LIN{ E6POS: X 709.1620, Y 12.2455, Z -112.0150, A 0, B 90, C 0, E1 0, E2 0, E3 0, E4 0 } C_DIS
LIN{ E6POS: X 709.1855, Y 12.9576, Z -112.0150, A 0, B 90, C 0, E1 0, E2 0, E3 0, E4 0 } C_DIS
LIN{ E6POS: X 709.1944, Y 13.6424, Z -112.0150, A 0, B 90, C 0, E1 0, E2 0, E3 0, E4 0 } C_DIS
LIN{ E6POS: X 709.2185, Y 14.3759, Z -112.0150, A 0, B 90, C 0, E1 0, E2 0, E3 0, E4 0 } C_DIS
LIN{ E6POS: X 709.2277, Y 15.0601, Z -112.0150, A 0, B 90, C 0, E1 0, E2 0, E3 0, E4 0 } C_DIS
LIN{ E6POS: X 709.2521, Y 15.7930, Z -112.0150, A 0, B 90, C 0, E1 0, E2 0, E3 0, E4 0 } C_DIS
LIN{ E6POS: X 709.2586, Y 16.4546, Z -112.0150, A 0, B 90, C 0, E1 0, E2 0, E3 0, E4 0 } C_DIS
LIN{ E6POS: X 709.2824, Y 17.1639, Z -112.0150, A 0, B 90, C 0, E1 0, E2 0, E3 0, E4 0 } C_DIS
LIN{ E6POS: X 709.2841, Y 17.7821, Z -112.0150, A 0, B 90, C 0, E1 0, E2 0, E3 0, E4 0 } C_DIS
LIN{ E6POS: X 709.3065, Y 18.4443, Z -112.0150, A 0, B 90, C 0, E1 0, E2 0, E3 0, E4 0 } C_DIS
LIN{ E6POS: X 709.3061, Y 19.0402, Z -112.0150, A 0, B 90, C 0, E1 0, E2 0, E3 0, E4 0 } C_DIS
LIN{ E6POS: X 709.3272, Y 19.6784, Z -112.0150, A 0, B 90, C 0, E1 0, E2 0, E3 0, E4 0 } C_DIS
LIN{ E6POS: X 709.3275, Y 20.2736, Z -112.0150, A 0, B 90, C 0, E1 0, E2 0, E3 0, E4 0 } C_DIS
LIN{ E6POS: X 709.3493, Y 20.9106, Z -112.0150, A 0, B 90, C 0, E1 0, E2 0, E3 0, E4 0 } C_DIS
LIN{ E6POS: X 709.3528, Y 21.5252, Z -112.0150, A 0, B 90, C 0, E1 0, E2 0, E3 0, E4 0 } C_DIS
LIN{ E6POS: X 709.3767, Y 22.1837, Z -112.0150, A 0, B 90, C 0, E1 0, E2 0, E3 0, E4 0 } C_DIS
LIN{ E6POS: X 709.3863, Y 22.8398, Z -112.0150, A 0, B 90, C 0, E1 0, E2 0, E3 0, E4 0 } C_DIS
LIN{ E6POS: X 709.4122, Y 23.5420, Z -112.0150, A 0, B 90, C 0, E1 0, E2 0, E3 0, E4 0 } C_DIS
LIN{ E6POS: X 709.4258, Y 24.1924, Z -112.0150, A 0, B 90, C 0, E1 0, E2 0, E3 0, E4 0 } C_DIS
LIN{ E6POS: X 709.4549, Y 24.8978, Z -112.0150, A 0, B 90, C 0, E1 0, E2 0, E3 0, E4 0 } C_DIS
LIN{ E6POS: X 709.4716, Y 25.4954, Z -112.0150, A 0, B 90, C 0, E1 0, E2 0, E3 0, E4 0 } C_DIS
LIN{ E6POS: X 709.5021, Y 26.1621, Z -112.0150, A 0, B 90, C 0, E1 0, E2 0, E3 0, E4 0 } C_DIS
LIN{ E6POS: X 709.5463, Y 27.1611, Z -112.0150, A 0, B 90, C 0, E1 0, E2 0, E3 0, E4 0 } C_DIS
LIN{ E6POS: X 709.5464, Y 27.1641, Z -112.0150, A 0, B 90, C 0, E1 0, E2 0, E3 0, E4 0 } C_DIS
LIN{ E6POS: X 709.6142, Y 28.1618, Z -112.0150, A 0, B 90, C 0, E1 0, E2 0, E3 0, E4 0 } C_DIS
LIN{ E6POS: X 709.6325, Y 28.4296, Z -112.0150, A 0, B 90, C 0, E1 0, E2 0, E3 0, E4 0 } C_DIS
LIN{ E6POS: X 709.6724, Y 29.4288, Z -112.0150, A 0, B 90, C 0, E1 0, E2 0, E3 0, E4 0 } C_DIS
LIN{ E6POS: X 709.6727, Y 29.4368, Z -112.0150, A 0, B 90, C 0, E1 0, E2 0, E3 0, E4 0 } C_DIS
LIN{ E6POS: X 709.7423, Y 30.4344, Z -112.0150, A 0, B 90, C 0, E1 0, E2 0, E3 0, E4 0 } C_DIS
LIN{ E6POS: X 709.7598, Y 30.6853, Z -112.0150, A 0, B 90, C 0, E1 0, E2 0, E3 0, E4 0 } C_DIS
LIN{ E6POS: X 709.7733, Y 31.4340, Z -112.0150, A 0, B 90, C 0, E1 0, E2 0, E3 0, E4 0 } C_DIS
LIN{ E6POS: X 709.8048, Y 32.1998, Z -112.0150, A 0, B 90, C 0, E1 0, E2 0, E3 0, E4 0 } C_DIS
LIN{ E6POS: X 709.8180, Y 33.0718, Z -112.0150, A 0, B 90, C 0, E1 0, E2 0, E3 0, E4 0 } C_DIS
LIN{ E6POS: X 709.8486, Y 33.9336, Z -112.0150, A 0, B 90, C 0, E1 0, E2 0, E3 0, E4 0 } C_DIS
LIN{ E6POS: X 709.8618, Y 34.8057, Z -112.0150, A 0, B 90, C 0, E1 0, E2 0, E3 0, E4 0 } C_DIS
LIN{ E6POS: X 709.8928, Y 35.6668, Z -112.0150, A 0, B 90, C 0, E1 0, E2 0, E3 0, E4 0 } C_DIS
LIN{ E6POS: X 709.9072, Y 36.4152, Z -112.0150, A 0, B 90, C 0, E1 0, E2 0, E3 0, E4 0 } C_DIS
LIN{ E6POS: X 709.9403, Y 37.1800, Z -112.0150, A 0, B 90, C 0, E1 0, E2 0, E3 0, E4 0 } C_DIS
LIN{ E6POS: X 709.9764, Y 38.0568, Z -112.0150, A 0, B 90, C 0, E1 0, E2 0, E3 0, E4 0 } C_DIS
LIN{ E6POS: X 710.0507, Y 39.0541, Z -112.0150, A 0, B 90, C 0, E1 0, E2 0, E3 0, E4 0 } C_DIS
LIN{ E6POS: X 710.0543, Y 39.1022, Z -112.0150, A 0, B 90, C 0, E1 0, E2 0, E3 0, E4 0 } C_DIS
LIN{ E6POS: X 710.1008, Y 39.9703, Z -112.0150, A 0, B 90, C 0, E1 0, E2 0, E3 0, E4 0 } C_DIS
LIN{ E6POS: X 710.1840, Y 40.9668, Z -112.0150, A 0, B 90, C 0, E1 0, E2 0, E3 0, E4 0 } C_DIS
LIN{ E6POS: X 710.1874, Y 41.0075, Z -112.0150, A 0, B 90, C 0, E1 0, E2 0, E3 0, E4 0 } C_DIS
LIN{ E6POS: X 710.2166, Y 41.7433, Z -112.0150, A 0, B 90, C 0, E1 0, E2 0, E3 0, E4 0 } C_DIS
LIN{ E6POS: X 710.2637, Y 42.4956, Z -112.0150, A 0, B 90, C 0, E1 0, E2 0, E3 0, E4 0 } C_DIS
LIN{ E6POS: X 710.2954, Y 43.3763, Z -112.0150, A 0, B 90, C 0, E1 0, E2 0, E3 0, E4 0 } C_DIS
LIN{ E6POS: X 710.3438, Y 44.2406, Z -112.0150, A 0, B 90, C 0, E1 0, E2 0, E3 0, E4 0 } C_DIS
LIN{ E6POS: X 710.3760, Y 45.1706, Z -112.0150, A 0, B 90, C 0, E1 0, E2 0, E3 0, E4 0 } C_DIS
LIN{ E6POS: X 710.4250, Y 46.0693, Z -112.0150, A 0, B 90, C 0, E1 0, E2 0, E3 0, E4 0 } C_DIS
LIN{ E6POS: X 710.4558, Y 46.9518, Z -112.0150, A 0, B 90, C 0, E1 0, E2 0, E3 0, E4 0 } C_DIS
LIN{ E6POS: X 710.5046, Y 47.8100, Z -112.0150, A 0, B 90, C 0, E1 0, E2 0, E3 0, E4 0 } C_DIS
LIN{ E6POS: X 710.5328, Y 48.5487, Z -112.0150, A 0, B 90, C 0, E1 0, E2 0, E3 0, E4 0 } C_DIS
LIN{ E6POS: X 710.5811, Y 49.2887, Z -112.0150, A 0, B 90, C 0, E1 0, E2 0, E3 0, E4 0 } C_DIS
LIN{ E6POS: X 710.6062, Y 49.9190, Z -112.0150, A 0, B 90, C 0, E1 0, E2 0, E3 0, E4 0 } C_DIS
LIN{ E6POS: X 710.6544, Y 50.5709, Z -112.0150, A 0, B 90, C 0, E1 0, E2 0, E3 0, E4 0 } C_DIS
LIN{ E6POS: X 710.6788, Y 51.1296, Z -112.0150, A 0, B 90, C 0, E1 0, E2 0, E3 0, E4 0 } C_DIS
LIN{ E6POS: X 710.7266, Y 51.7228, Z -112.0150, A 0, B 90, C 0, E1 0, E2 0, E3 0, E4 0 } C_DIS
LIN{ E6POS: X 710.7500, Y 52.2478, Z -112.0150, A 0, B 90, C 0, E1 0, E2 0, E3 0, E4 0 } C_DIS
LIN{ E6POS: X 710.7981, Y 52.8176, Z -112.0150, A 0, B 90, C 0, E1 0, E2 0, E3 0, E4 0 } C_DIS
LIN{ E6POS: X 711.3004, Y 52.6997, Z -112.0150, A 0, B 90, C 0, E1 0, E2 0, E3 0, E4 0 } C_DIS
LIN{ E6POS: X 711.8008, Y 52.5905, Z -112.0150, A 0, B 90, C 0, E1 0, E2 0, E3 0, E4 0 } C_DIS
LIN{ E6POS: X 712.7693, Y 52.3414, Z -112.0150, A 0, B 90, C 0, E1 0, E2 0, E3 0, E4 0 } C_DIS
LIN{ E6POS: X 713.3037, Y 52.2039, Z -112.0150, A 0, B 90, C 0, E1 0, E2 0, E3 0, E4 0 } C_DIS
LIN{ E6POS: X 714.2696, Y 51.9451, Z -112.0150, A 0, B 90, C 0, E1 0, E2 0, E3 0, E4 0 } C_DIS
LIN{ E6POS: X 714.7957, Y 51.8041, Z -112.0150, A 0, B 90, C 0, E1 0, E2 0, E3 0, E4 0 } C_DIS
LIN{ E6POS: X 715.7636, Y 51.5525, Z -112.0150, A 0, B 90, C 0, E1 0, E2 0, E3 0, E4 0 } C_DIS
LIN{ E6POS: X 716.7314, Y 51.3008, Z -112.0150, A 0, B 90, C 0, E1 0, E2 0, E3 0, E4 0 } C_DIS
LIN{ E6POS: X 717.6992, Y 51.0492, Z -112.0150, A 0, B 90, C 0, E1 0, E2 0, E3 0, E4 0 } C_DIS
LIN{ E6POS: X 717.8000, Y 51.0230, Z -112.0150, A 0, B 90, C 0, E1 0, E2 0, E3 0, E4 0 } C_DIS
LIN{ E6POS: X 718.7644, Y 50.7585, Z -112.0150, A 0, B 90, C 0, E1 0, E2 0, E3 0, E4 0 } C_DIS
LIN{ E6POS: X 719.7288, Y 50.4939, Z -112.0150, A 0, B 90, C 0, E1 0, E2 0, E3 0, E4 0 } C_DIS
LIN{ E6POS: X 720.6931, Y 50.2294, Z -112.0150, A 0, B 90, C 0, E1 0, E2 0, E3 0, E4 0 } C_DIS
LIN{ E6POS: X 720.7818, Y 50.2051, Z -112.0150, A 0, B 90, C 0, E1 0, E2 0, E3 0, E4 0 } C_DIS
LIN{ E6POS: X 721.7493, Y 49.9525, Z -112.0150, A 0, B 90, C 0, E1 0, E2 0, E3 0, E4 0 } C_DIS
LIN{ E6POS: X 722.7169, Y 49.6999, Z -112.0150, A 0, B 90, C 0, E1 0, E2 0, E3 0, E4 0 } C_DIS
LIN{ E6POS: X 723.6845, Y 49.4472, Z -112.0150, A 0, B 90, C 0, E1 0, E2 0, E3 0, E4 0 } C_DIS
LIN{ E6POS: X 724.6520, Y 49.1946, Z -112.0150, A 0, B 90, C 0, E1 0, E2 0, E3 0, E4 0 } C_DIS
LIN{ E6POS: X 725.6196, Y 48.9420, Z -112.0150, A 0, B 90, C 0, E1 0, E2 0, E3 0, E4 0 } C_DIS
LIN{ E6POS: X 725.7889, Y 48.8978, Z -112.0150, A 0, B 90, C 0, E1 0, E2 0, E3 0, E4 0 } C_DIS
LIN{ E6POS: X 726.7527, Y 48.6312, Z -112.0150, A 0, B 90, C 0, E1 0, E2 0, E3 0, E4 0 } C_DIS
LIN{ E6POS: X 727.7165, Y 48.3646, Z -112.0150, A 0, B 90, C 0, E1 0, E2 0, E3 0, E4 0 } C_DIS
LIN{ E6POS: X 728.6803, Y 48.0980, Z -112.0150, A 0, B 90, C 0, E1 0, E2 0, E3 0, E4 0 } C_DIS
LIN{ E6POS: X 729.6441, Y 47.8314, Z -112.0150, A 0, B 90, C 0, E1 0, E2 0, E3 0, E4 0 } C_DIS
LIN{ E6POS: X 730.6079, Y 47.5648, Z -112.0150, A 0, B 90, C 0, E1 0, E2 0, E3 0, E4 0 } C_DIS
LIN{ E6POS: X 730.7577, Y 47.5233, Z -112.0150, A 0, B 90, C 0, E1 0, E2 0, E3 0, E4 0 } C_DIS
LIN{ E6POS: X 731.7278, Y 47.2808, Z -112.0150, A 0, B 90, C 0, E1 0, E2 0, E3 0, E4 0 } C_DIS
LIN{ E6POS: X 732.6980, Y 47.0382, Z -112.0150, A 0, B 90, C 0, E1 0, E2 0, E3 0, E4 0 } C_DIS
LIN{ E6POS: X 733.6681, Y 46.7957, Z -112.0150, A 0, B 90, C 0, E1 0, E2 0, E3 0, E4 0 } C_DIS
LIN{ E6POS: X 734.6382, Y 46.5532, Z -112.0150, A 0, B 90, C 0, E1 0, E2 0, E3 0, E4 0 } C_DIS
LIN{ E6POS: X 735.6084, Y 46.3106, Z -112.0150, A 0, B 90, C 0, E1 0, E2 0, E3 0, E4 0 } C_DIS
LIN{ E6POS: X 736.5785, Y 46.0681, Z -112.0150, A 0, B 90, C 0, E1 0, E2 0, E3 0, E4 0 } C_DIS
LIN{ E6POS: X 736.9469, Y 45.9760, Z -112.0150, A 0, B 90, C 0, E1 0, E2 0, E3 0, E4 0 } C_DIS
LIN{ E6POS: X 737.9136, Y 45.7202, Z -112.0150, A 0, B 90, C 0, E1 0, E2 0, E3 0, E4 0 } C_DIS
LIN{ E6POS: X 738.8803, Y 45.4644, Z -112.0150, A 0, B 90, C 0, E1 0, E2 0, E3 0, E4 0 } C_DIS
LIN{ E6POS: X 739.8471, Y 45.2087, Z -112.0150, A 0, B 90, C 0, E1 0, E2 0, E3 0, E4 0 } C_DIS
LIN{ E6POS: X 740.8138, Y 44.9529, Z -112.0150, A 0, B 90, C 0, E1 0, E2 0, E3 0, E4 0 } C_DIS
LIN{ E6POS: X 741.7806, Y 44.6971, Z -112.0150, A 0, B 90, C 0, E1 0, E2 0, E3 0, E4 0 } C_DIS
LIN{ E6POS: X 742.7473, Y 44.4414, Z -112.0150, A 0, B 90, C 0, E1 0, E2 0, E3 0, E4 0 } C_DIS
LIN{ E6POS: X 743.1041, Y 44.3470, Z -112.0150, A 0, B 90, C 0, E1 0, E2 0, E3 0, E4 0 } C_DIS
LIN{ E6POS: X 744.0789, Y 44.1236, Z -112.0150, A 0, B 90, C 0, E1 0, E2 0, E3 0, E4 0 } C_DIS
LIN{ E6POS: X 745.0536, Y 43.9003, Z -112.0150, A 0, B 90, C 0, E1 0, E2 0, E3 0, E4 0 } C_DIS
LIN{ E6POS: X 746.0283, Y 43.6769, Z -112.0150, A 0, B 90, C 0, E1 0, E2 0, E3 0, E4 0 } C_DIS
LIN{ E6POS: X 747.0031, Y 43.4536, Z -112.0150, A 0, B 90, C 0, E1 0, E2 0, E3 0, E4 0 } C_DIS
LIN{ E6POS: X 747.9778, Y 43.2302, Z -112.0150, A 0, B 90, C 0, E1 0, E2 0, E3 0, E4 0 } C_DIS
LIN{ E6POS: X 748.9526, Y 43.0068, Z -112.0150, A 0, B 90, C 0, E1 0, E2 0, E3 0, E4 0 } C_DIS
LIN{ E6POS: X 749.6560, Y 42.8457, Z -112.0150, A 0, B 90, C 0, E1 0, E2 0, E3 0, E4 0 } C_DIS
LIN{ E6POS: X 750.6282, Y 42.6112, Z -112.0150, A 0, B 90, C 0, E1 0, E2 0, E3 0, E4 0 } C_DIS
LIN{ E6POS: X 751.6003, Y 42.3768, Z -112.0150, A 0, B 90, C 0, E1 0, E2 0, E3 0, E4 0 } C_DIS
LIN{ E6POS: X 752.5724, Y 42.1423, Z -112.0150, A 0, B 90, C 0, E1 0, E2 0, E3 0, E4 0 } C_DIS
LIN{ E6POS: X 753.5445, Y 41.9079, Z -112.0150, A 0, B 90, C 0, E1 0, E2 0, E3 0, E4 0 } C_DIS
LIN{ E6POS: X 754.5167, Y 41.6734, Z -112.0150, A 0, B 90, C 0, E1 0, E2 0, E3 0, E4 0 } C_DIS
LIN{ E6POS: X 755.4888, Y 41.4390, Z -112.0150, A 0, B 90, C 0, E1 0, E2 0, E3 0, E4 0 } C_DIS
LIN{ E6POS: X 756.2065, Y 41.2659, Z -112.0150, A 0, B 90, C 0, E1 0, E2 0, E3 0, E4 0 } C_DIS
LIN{ E6POS: X 757.1886, Y 41.0774, Z -112.0150, A 0, B 90, C 0, E1 0, E2 0, E3 0, E4 0 } C_DIS
LIN{ E6POS: X 758.1707, Y 40.8890, Z -112.0150, A 0, B 90, C 0, E1 0, E2 0, E3 0, E4 0 } C_DIS
LIN{ E6POS: X 759.1528, Y 40.7006, Z -112.0150, A 0, B 90, C 0, E1 0, E2 0, E3 0, E4 0 } C_DIS
LIN{ E6POS: X 760.1349, Y 40.5122, Z -112.0150, A 0, B 90, C 0, E1 0, E2 0, E3 0, E4 0 } C_DIS
LIN{ E6POS: X 761.1170, Y 40.3237, Z -112.0150, A 0, B 90, C 0, E1 0, E2 0, E3 0, E4 0 } C_DIS
LIN{ E6POS: X 762.0991, Y 40.1353, Z -112.0150, A 0, B 90, C 0, E1 0, E2 0, E3 0, E4 0 } C_DIS
LIN{ E6POS: X 762.3004, Y 40.0967, Z -112.0150, A 0, B 90, C 0, E1 0, E2 0, E3 0, E4 0 } C_DIS
LIN{ E6POS: X 763.2810, Y 39.9006, Z -112.0150, A 0, B 90, C 0, E1 0, E2 0, E3 0, E4 0 } C_DIS
LIN{ E6POS: X 764.2616, Y 39.7046, Z -112.0150, A 0, B 90, C 0, E1 0, E2 0, E3 0, E4 0 } C_DIS
LIN{ E6POS: X 765.2422, Y 39.5086, Z -112.0150, A 0, B 90, C 0, E1 0, E2 0, E3 0, E4 0 } C_DIS
LIN{ E6POS: X 766.2228, Y 39.3125, Z -112.0150, A 0, B 90, C 0, E1 0, E2 0, E3 0, E4 0 } C_DIS
LIN{ E6POS: X 767.2034, Y 39.1165, Z -112.0150, A 0, B 90, C 0, E1 0, E2 0, E3 0, E4 0 } C_DIS
LIN{ E6POS: X 768.1840, Y 38.9204, Z -112.0150, A 0, B 90, C 0, E1 0, E2 0, E3 0, E4 0 } C_DIS
LIN{ E6POS: X 768.4460, Y 38.8681, Z -112.0150, A 0, B 90, C 0, E1 0, E2 0, E3 0, E4 0 } C_DIS
LIN{ E6POS: X 769.4396, Y 38.7544, Z -112.0150, A 0, B 90, C 0, E1 0, E2 0, E3 0, E4 0 } C_DIS
LIN{ E6POS: X 770.4331, Y 38.6408, Z -112.0150, A 0, B 90, C 0, E1 0, E2 0, E3 0, E4 0 } C_DIS
LIN{ E6POS: X 771.4266, Y 38.5271, Z -112.0150, A 0, B 90, C 0, E1 0, E2 0, E3 0, E4 0 } C_DIS
LIN{ E6POS: X 772.4201, Y 38.4135, Z -112.0150, A 0, B 90, C 0, E1 0, E2 0, E3 0, E4 0 } C_DIS
LIN{ E6POS: X 773.2625, Y 38.3171, Z -112.0150, A 0, B 90, C 0, E1 0, E2 0, E3 0, E4 0 } C_DIS
LIN{ E6POS: X 774.2558, Y 38.2019, Z -112.0150, A 0, B 90, C 0, E1 0, E2 0, E3 0, E4 0 } C_DIS
LIN{ E6POS: X 775.2492, Y 38.0868, Z -112.0150, A 0, B 90, C 0, E1 0, E2 0, E3 0, E4 0 } C_DIS
LIN{ E6POS: X 776.2425, Y 37.9716, Z -112.0150, A 0, B 90, C 0, E1 0, E2 0, E3 0, E4 0 } C_DIS
LIN{ E6POS: X 777.2359, Y 37.8565, Z -112.0150, A 0, B 90, C 0, E1 0, E2 0, E3 0, E4 0 } C_DIS
LIN{ E6POS: X 778.2062, Y 37.7440, Z -112.0150, A 0, B 90, C 0, E1 0, E2 0, E3 0, E4 0 } C_DIS
LIN{ E6POS: X 779.2060, Y 37.7214, Z -112.0150, A 0, B 90, C 0, E1 0, E2 0, E3 0, E4 0 } C_DIS
LIN{ E6POS: X 780.2057, Y 37.6989, Z -112.0150, A 0, B 90, C 0, E1 0, E2 0, E3 0, E4 0 } C_DIS
LIN{ E6POS: X 781.2055, Y 37.6763, Z -112.0150, A 0, B 90, C 0, E1 0, E2 0, E3 0, E4 0 } C_DIS
LIN{ E6POS: X 782.0641, Y 37.6570, Z -112.0150, A 0, B 90, C 0, E1 0, E2 0, E3 0, E4 0 } C_DIS
LIN{ E6POS: X 783.0639, Y 37.6365, Z -112.0150, A 0, B 90, C 0, E1 0, E2 0, E3 0, E4 0 } C_DIS
LIN{ E6POS: X 784.0637, Y 37.6161, Z -112.0150, A 0, B 90, C 0, E1 0, E2 0, E3 0, E4 0 } C_DIS
LIN{ E6POS: X 785.0635, Y 37.5956, Z -112.0150, A 0, B 90, C 0, E1 0, E2 0, E3 0, E4 0 } C_DIS
LIN{ E6POS: X 786.0633, Y 37.5751, Z -112.0150, A 0, B 90, C 0, E1 0, E2 0, E3 0, E4 0 } C_DIS
LIN{ E6POS: X 786.1069, Y 37.5742, Z -112.0150, A 0, B 90, C 0, E1 0, E2 0, E3 0, E4 0 } C_DIS
LIN{ E6POS: X 787.1045, Y 37.6431, Z -112.0150, A 0, B 90, C 0, E1 0, E2 0, E3 0, E4 0 } C_DIS
LIN{ E6POS: X 788.1021, Y 37.7120, Z -112.0150, A 0, B 90, C 0, E1 0, E2 0, E3 0, E4 0 } C_DIS
LIN{ E6POS: X 789.0998, Y 37.7809, Z -112.0150, A 0, B 90, C 0, E1 0, E2 0, E3 0, E4 0 } C_DIS
LIN{ E6POS: X 789.3264, Y 37.7965, Z -112.0150, A 0, B 90, C 0, E1 0, E2 0, E3 0, E4 0 } C_DIS
LIN{ E6POS: X 790.3238, Y 37.8673, Z -112.0150, A 0, B 90, C 0, E1 0, E2 0, E3 0, E4 0 } C_DIS
LIN{ E6POS: X 791.3213, Y 37.9382, Z -112.0150, A 0, B 90, C 0, E1 0, E2 0, E3 0, E4 0 } C_DIS
LIN{ E6POS: X 792.3188, Y 38.0090, Z -112.0150, A 0, B 90, C 0, E1 0, E2 0, E3 0, E4 0 } C_DIS
LIN{ E6POS: X 792.7685, Y 38.0409, Z -112.0150, A 0, B 90, C 0, E1 0, E2 0, E3 0, E4 0 } C_DIS
LIN{ E6POS: X 793.7601, Y 38.1698, Z -112.0150, A 0, B 90, C 0, E1 0, E2 0, E3 0, E4 0 } C_DIS
LIN{ E6POS: X 794.7518, Y 38.2986, Z -112.0150, A 0, B 90, C 0, E1 0, E2 0, E3 0, E4 0 } C_DIS
LIN{ E6POS: X 795.6682, Y 38.4177, Z -112.0150, A 0, B 90, C 0, E1 0, E2 0, E3 0, E4 0 } C_DIS
LIN{ E6POS: X 796.6599, Y 38.5466, Z -112.0150, A 0, B 90, C 0, E1 0, E2 0, E3 0, E4 0 } C_DIS
LIN{ E6POS: X 797.6516, Y 38.6755, Z -112.0150, A 0, B 90, C 0, E1 0, E2 0, E3 0, E4 0 } C_DIS
LIN{ E6POS: X 798.6432, Y 38.8044, Z -112.0150, A 0, B 90, C 0, E1 0, E2 0, E3 0, E4 0 } C_DIS
LIN{ E6POS: X 798.8097, Y 38.8260, Z -112.0150, A 0, B 90, C 0, E1 0, E2 0, E3 0, E4 0 } C_DIS
LIN{ E6POS: X 798.7068, Y 37.8313, Z -112.0150, A 0, B 90, C 0, E1 0, E2 0, E3 0, E4 0 } C_DIS
LIN{ E6POS: X 798.6040, Y 36.8366, Z -112.0150, A 0, B 90, C 0, E1 0, E2 0, E3 0, E4 0 } C_DIS
LIN{ E6POS: X 798.5012, Y 35.8419, Z -112.0150, A 0, B 90, C 0, E1 0, E2 0, E3 0, E4 0 } C_DIS
LIN{ E6POS: X 798.3983, Y 34.8472, Z -112.0150, A 0, B 90, C 0, E1 0, E2 0, E3 0, E4 0 } C_DIS
LIN{ E6POS: X 798.2955, Y 33.8525, Z -112.0150, A 0, B 90, C 0, E1 0, E2 0, E3 0, E4 0 } C_DIS
LIN{ E6POS: X 798.1927, Y 32.8578, Z -112.0150, A 0, B 90, C 0, E1 0, E2 0, E3 0, E4 0 } C_DIS
LIN{ E6POS: X 798.0898, Y 31.8631, Z -112.0150, A 0, B 90, C 0, E1 0, E2 0, E3 0, E4 0 } C_DIS
LIN{ E6POS: X 797.9998, Y 30.9920, Z -112.0150, A 0, B 90, C 0, E1 0, E2 0, E3 0, E4 0 } C_DIS
LIN{ E6POS: X 797.8969, Y 29.9973, Z -112.0150, A 0, B 90, C 0, E1 0, E2 0, E3 0, E4 0 } C_DIS
LIN{ E6POS: X 797.7941, Y 29.0026, Z -112.0150, A 0, B 90, C 0, E1 0, E2 0, E3 0, E4 0 } C_DIS
LIN{ E6POS: X 797.6913, Y 28.0079, Z -112.0150, A 0, B 90, C 0, E1 0, E2 0, E3 0, E4 0 } C_DIS
LIN{ E6POS: X 797.5884, Y 27.0132, Z -112.0150, A 0, B 90, C 0, E1 0, E2 0, E3 0, E4 0 } C_DIS
LIN{ E6POS: X 797.4856, Y 26.0185, Z -112.0150, A 0, B 90, C 0, E1 0, E2 0, E3 0, E4 0 } C_DIS
LIN{ E6POS: X 797.3828, Y 25.0238, Z -112.0150, A 0, B 90, C 0, E1 0, E2 0, E3 0, E4 0 } C_DIS
LIN{ E6POS: X 797.2799, Y 24.0291, Z -112.0150, A 0, B 90, C 0, E1 0, E2 0, E3 0, E4 0 } C_DIS
LIN{ E6POS: X 797.1771, Y 23.0344, Z -112.0150, A 0, B 90, C 0, E1 0, E2 0, E3 0, E4 0 } C_DIS
LIN{ E6POS: X 797.1224, Y 22.5051, Z -110.0150, A 0, B 90, C 0, E1 0, E2 0, E3 0, E4 0 } C_DIS
LIN{ E6POS: X 797.0002, Y 21.5126, Z -110.0150, A 0, B 90, C 0, E1 0, E2 0, E3 0, E4 0 } C_DIS
LIN{ E6POS: X 796.8780, Y 20.5201, Z -110.0150, A 0, B 90, C 0, E1 0, E2 0, E3 0, E4 0 } C_DIS
LIN{ E6POS: X 796.7559, Y 19.5276, Z -110.0150, A 0, B 90, C 0, E1 0, E2 0, E3 0, E4 0 } C_DIS
LIN{ E6POS: X 796.6337, Y 18.5351, Z -110.0150, A 0, B 90, C 0, E1 0, E2 0, E3 0, E4 0 } C_DIS
LIN{ E6POS: X 796.5115, Y 17.5426, Z -110.0150, A 0, B 90, C 0, E1 0, E2 0, E3 0, E4 0 } C_DIS
LIN{ E6POS: X 796.3893, Y 16.5500, Z -110.0150, A 0, B 90, C 0, E1 0, E2 0, E3 0, E4 0 } C_DIS
LIN{ E6POS: X 796.2672, Y 15.5575, Z -110.0150, A 0, B 90, C 0, E1 0, E2 0, E3 0, E4 0 } C_DIS
LIN{ E6POS: X 796.1450, Y 14.5650, Z -110.0150, A 0, B 90, C 0, E1 0, E2 0, E3 0, E4 0 } C_DIS
LIN{ E6POS: X 796.0773, Y 14.0156, Z -110.0150, A 0, B 90, C 0, E1 0, E2 0, E3 0, E4 0 } C_DIS
LIN{ E6POS: X 795.9552, Y 13.0231, Z -110.0150, A 0, B 90, C 0, E1 0, E2 0, E3 0, E4 0 } C_DIS
LIN{ E6POS: X 795.8330, Y 12.0306, Z -110.0150, A 0, B 90, C 0, E1 0, E2 0, E3 0, E4 0 } C_DIS
LIN{ E6POS: X 795.7108, Y 11.0381, Z -110.0150, A 0, B 90, C 0, E1 0, E2 0, E3 0, E4 0 } C_DIS
LIN{ E6POS: X 795.5886, Y 10.0455, Z -110.0150, A 0, B 90, C 0, E1 0, E2 0, E3 0, E4 0 } C_DIS
LIN{ E6POS: X 795.4665, Y 9.0530, Z -110.0150, A 0, B 90, C 0, E1 0, E2 0, E3 0, E4 0 } C_DIS
LIN{ E6POS: X 795.3443, Y 8.0605, Z -110.0150, A 0, B 90, C 0, E1 0, E2 0, E3 0, E4 0 } C_DIS
LIN{ E6POS: X 795.2562, Y 7.3452, Z -110.0150, A 0, B 90, C 0, E1 0, E2 0, E3 0, E4 0 } C_DIS
LIN{ E6POS: X 795.0854, Y 6.3599, Z -110.0150, A 0, B 90, C 0, E1 0, E2 0, E3 0, E4 0 } C_DIS
LIN{ E6POS: X 794.9146, Y 5.3746, Z -110.0150, A 0, B 90, C 0, E1 0, E2 0, E3 0, E4 0 } C_DIS
LIN{ E6POS: X 794.7438, Y 4.3893, Z -110.0150, A 0, B 90, C 0, E1 0, E2 0, E3 0, E4 0 } C_DIS
LIN{ E6POS: X 794.5730, Y 3.4040, Z -110.0150, A 0, B 90, C 0, E1 0, E2 0, E3 0, E4 0 } C_DIS
LIN{ E6POS: X 794.4021, Y 2.4187, Z -110.0150, A 0, B 90, C 0, E1 0, E2 0, E3 0, E4 0 } C_DIS
LIN{ E6POS: X 794.2313, Y 1.4334, Z -110.0150, A 0, B 90, C 0, E1 0, E2 0, E3 0, E4 0 } C_DIS
LIN{ E6POS: X 794.0605, Y 0.4481, Z -110.0150, A 0, B 90, C 0, E1 0, E2 0, E3 0, E4 0 } C_DIS
LIN{ E6POS: X 794.0101, Y 0.1575, Z -110.0150, A 0, B 90, C 0, E1 0, E2 0, E3 0, E4 0 } C_DIS
LIN{ E6POS: X 793.8393, Y -0.8278, Z -110.0150, A 0, B 90, C 0, E1 0, E2 0, E3 0, E4 0 } C_DIS
LIN{ E6POS: X 793.6685, Y -1.8131, Z -110.0150, A 0, B 90, C 0, E1 0, E2 0, E3 0, E4 0 } C_DIS
LIN{ E6POS: X 793.4977, Y -2.7984, Z -110.0150, A 0, B 90, C 0, E1 0, E2 0, E3 0, E4 0 } C_DIS
LIN{ E6POS: X 793.3268, Y -3.7837, Z -110.0150, A 0, B 90, C 0, E1 0, E2 0, E3 0, E4 0 } C_DIS
LIN{ E6POS: X 793.1560, Y -4.7690, Z -110.0150, A 0, B 90, C 0, E1 0, E2 0, E3 0, E4 0 } C_DIS
LIN{ E6POS: X 793.0310, Y -5.4900, Z -110.0150, A 0, B 90, C 0, E1 0, E2 0, E3 0, E4 0 } C_DIS
LIN{ E6POS: X 792.7476, Y -6.4490, Z -110.0150, A 0, B 90, C 0, E1 0, E2 0, E3 0, E4 0 } C_DIS
LIN{ E6POS: X 792.4642, Y -7.4080, Z -110.0150, A 0, B 90, C 0, E1 0, E2 0, E3 0, E4 0 } C_DIS
LIN{ E6POS: X 792.1808, Y -8.3670, Z -110.0150, A 0, B 90, C 0, E1 0, E2 0, E3 0, E4 0 } C_DIS
LIN{ E6POS: X 791.8974, Y -9.3260, Z -110.0150, A 0, B 90, C 0, E1 0, E2 0, E3 0, E4 0 } C_DIS
LIN{ E6POS: X 791.6139, Y -10.2850, Z -110.0150, A 0, B 90, C 0, E1 0, E2 0, E3 0, E4 0 } C_DIS
LIN{ E6POS: X 791.4838, Y -10.7253, Z -110.0150, A 0, B 90, C 0, E1 0, E2 0, E3 0, E4 0 } C_DIS
LIN{ E6POS: X 791.2004, Y -11.6843, Z -110.0150, A 0, B 90, C 0, E1 0, E2 0, E3 0, E4 0 } C_DIS
LIN{ E6POS: X 790.9170, Y -12.6433, Z -110.0150, A 0, B 90, C 0, E1 0, E2 0, E3 0, E4 0 } C_DIS
LIN{ E6POS: X 790.6336, Y -13.6023, Z -110.0150, A 0, B 90, C 0, E1 0, E2 0, E3 0, E4 0 } C_DIS
LIN{ E6POS: X 790.3501, Y -14.5613, Z -110.0150, A 0, B 90, C 0, E1 0, E2 0, E3 0, E4 0 } C_DIS
LIN{ E6POS: X 790.2681, Y -14.8387, Z -110.0150, A 0, B 90, C 0, E1 0, E2 0, E3 0, E4 0 } C_DIS
LIN{ E6POS: X 789.6733, Y -15.6426, Z -110.0150, A 0, B 90, C 0, E1 0, E2 0, E3 0, E4 0 } C_DIS
LIN{ E6POS: X 789.0784, Y -16.4464, Z -110.0150, A 0, B 90, C 0, E1 0, E2 0, E3 0, E4 0 } C_DIS
LIN{ E6POS: X 788.4835, Y -17.2502, Z -110.0150, A 0, B 90, C 0, E1 0, E2 0, E3 0, E4 0 } C_DIS
LIN{ E6POS: X 788.3195, Y -17.4719, Z -110.0150, A 0, B 90, C 0, E1 0, E2 0, E3 0, E4 0 } C_DIS
LIN{ E6POS: X 787.7246, Y -18.2757, Z -110.0150, A 0, B 90, C 0, E1 0, E2 0, E3 0, E4 0 } C_DIS
LIN{ E6POS: X 787.1298, Y -19.0795, Z -110.0150, A 0, B 90, C 0, E1 0, E2 0, E3 0, E4 0 } C_DIS
LIN{ E6POS: X 786.7884, Y -19.5408, Z -110.0150, A 0, B 90, C 0, E1 0, E2 0, E3 0, E4 0 } C_DIS
LIN{ E6POS: X 785.8312, Y -19.8300, Z -110.0150, A 0, B 90, C 0, E1 0, E2 0, E3 0, E4 0 } C_DIS
LIN{ E6POS: X 784.8739, Y -20.1192, Z -110.0150, A 0, B 90, C 0, E1 0, E2 0, E3 0, E4 0 } C_DIS
LIN{ E6POS: X 784.3102, Y -20.2895, Z -110.0150, A 0, B 90, C 0, E1 0, E2 0, E3 0, E4 0 } C_DIS
LIN{ E6POS: X 783.3541, Y -20.5827, Z -110.0150, A 0, B 90, C 0, E1 0, E2 0, E3 0, E4 0 } C_DIS
LIN{ E6POS: X 782.3980, Y -20.8758, Z -110.0150, A 0, B 90, C 0, E1 0, E2 0, E3 0, E4 0 } C_DIS
LIN{ E6POS: X 782.3889, Y -20.8786, Z -110.0150, A 0, B 90, C 0, E1 0, E2 0, E3 0, E4 0 } C_DIS
LIN{ E6POS: X 781.3980, Y -20.7437, Z -110.0150, A 0, B 90, C 0, E1 0, E2 0, E3 0, E4 0 } C_DIS
LIN{ E6POS: X 780.4071, Y -20.6088, Z -110.0150, A 0, B 90, C 0, E1 0, E2 0, E3 0, E4 0 } C_DIS
LIN{ E6POS: X 780.0031, Y -20.5538, Z -110.0150, A 0, B 90, C 0, E1 0, E2 0, E3 0, E4 0 } C_DIS
LIN{ E6POS: X 779.0117, Y -20.4222, Z -110.0150, A 0, B 90, C 0, E1 0, E2 0, E3 0, E4 0 } C_DIS
LIN{ E6POS: X 778.0204, Y -20.2906, Z -110.0150, A 0, B 90, C 0, E1 0, E2 0, E3 0, E4 0 } C_DIS
LIN{ E6POS: X 777.0291, Y -20.1589, Z -110.0150, A 0, B 90, C 0, E1 0, E2 0, E3 0, E4 0 } C_DIS
LIN{ E6POS: X 776.8686, Y -20.1376, Z -110.0150, A 0, B 90, C 0, E1 0, E2 0, E3 0, E4 0 } C_DIS
LIN{ E6POS: X 775.8941, Y -19.9135, Z -110.0150, A 0, B 90, C 0, E1 0, E2 0, E3 0, E4 0 } C_DIS
LIN{ E6POS: X 774.9195, Y -19.6894, Z -110.0150, A 0, B 90, C 0, E1 0, E2 0, E3 0, E4 0 } C_DIS
LIN{ E6POS: X 773.9449, Y -19.4654, Z -110.0150, A 0, B 90, C 0, E1 0, E2 0, E3 0, E4 0 } C_DIS
LIN{ E6POS: X 773.9439, Y -19.4651, Z -110.0150, A 0, B 90, C 0, E1 0, E2 0, E3 0, E4 0 } C_DIS
LIN{ E6POS: X 772.9673, Y -19.2503, Z -110.0150, A 0, B 90, C 0, E1 0, E2 0, E3 0, E4 0 } C_DIS
LIN{ E6POS: X 771.9907, Y -19.0354, Z -110.0150, A 0, B 90, C 0, E1 0, E2 0, E3 0, E4 0 } C_DIS
LIN{ E6POS: X 771.0140, Y -18.8205, Z -110.0150, A 0, B 90, C 0, E1 0, E2 0, E3 0, E4 0 } C_DIS
LIN{ E6POS: X 770.0374, Y -18.6056, Z -110.0150, A 0, B 90, C 0, E1 0, E2 0, E3 0, E4 0 } C_DIS
LIN{ E6POS: X 770.0249, Y -18.6029, Z -110.0150, A 0, B 90, C 0, E1 0, E2 0, E3 0, E4 0 } C_DIS
LIN{ E6POS: X 769.0331, Y -18.4752, Z -110.0150, A 0, B 90, C 0, E1 0, E2 0, E3 0, E4 0 } C_DIS
LIN{ E6POS: X 768.0412, Y -18.3476, Z -110.0150, A 0, B 90, C 0, E1 0, E2 0, E3 0, E4 0 } C_DIS
LIN{ E6POS: X 767.0494, Y -18.2199, Z -110.0150, A 0, B 90, C 0, E1 0, E2 0, E3 0, E4 0 } C_DIS
LIN{ E6POS: X 766.4865, Y -18.1475, Z -110.0150, A 0, B 90, C 0, E1 0, E2 0, E3 0, E4 0 } C_DIS
LIN{ E6POS: X 765.4938, Y -18.0263, Z -110.0150, A 0, B 90, C 0, E1 0, E2 0, E3 0, E4 0 } C_DIS
LIN{ E6POS: X 764.5012, Y -17.9052, Z -110.0150, A 0, B 90, C 0, E1 0, E2 0, E3 0, E4 0 } C_DIS
LIN{ E6POS: X 763.5086, Y -17.7840, Z -110.0150, A 0, B 90, C 0, E1 0, E2 0, E3 0, E4 0 } C_DIS
LIN{ E6POS: X 762.5159, Y -17.6629, Z -110.0150, A 0, B 90, C 0, E1 0, E2 0, E3 0, E4 0 } C_DIS
LIN{ E6POS: X 761.6559, Y -17.5579, Z -110.0150, A 0, B 90, C 0, E1 0, E2 0, E3 0, E4 0 } C_DIS
LIN{ E6POS: X 760.6582, Y -17.4908, Z -110.0150, A 0, B 90, C 0, E1 0, E2 0, E3 0, E4 0 } C_DIS
LIN{ E6POS: X 759.6604, Y -17.4237, Z -110.0150, A 0, B 90, C 0, E1 0, E2 0, E3 0, E4 0 } C_DIS
LIN{ E6POS: X 758.6627, Y -17.3566, Z -110.0150, A 0, B 90, C 0, E1 0, E2 0, E3 0, E4 0 } C_DIS
LIN{ E6POS: X 757.9358, Y -17.3077, Z -110.0150, A 0, B 90, C 0, E1 0, E2 0, E3 0, E4 0 } C_DIS
LIN{ E6POS: X 756.9379, Y -17.2430, Z -110.0150, A 0, B 90, C 0, E1 0, E2 0, E3 0, E4 0 } C_DIS
LIN{ E6POS: X 755.9400, Y -17.1782, Z -110.0150, A 0, B 90, C 0, E1 0, E2 0, E3 0, E4 0 } C_DIS
LIN{ E6POS: X 754.9421, Y -17.1135, Z -110.0150, A 0, B 90, C 0, E1 0, E2 0, E3 0, E4 0 } C_DIS
LIN{ E6POS: X 753.9442, Y -17.0488, Z -110.0150, A 0, B 90, C 0, E1 0, E2 0, E3 0, E4 0 } C_DIS
LIN{ E6POS: X 752.9463, Y -16.9840, Z -110.0150, A 0, B 90, C 0, E1 0, E2 0, E3 0, E4 0 } C_DIS
LIN{ E6POS: X 752.8087, Y -16.9751, Z -110.0150, A 0, B 90, C 0, E1 0, E2 0, E3 0, E4 0 } C_DIS
LIN{ E6POS: X 751.8088, Y -16.9588, Z -110.0150, A 0, B 90, C 0, E1 0, E2 0, E3 0, E4 0 } C_DIS
LIN{ E6POS: X 750.8089, Y -16.9426, Z -110.0150, A 0, B 90, C 0, E1 0, E2 0, E3 0, E4 0 } C_DIS
LIN{ E6POS: X 749.8090, Y -16.9263, Z -110.0150, A 0, B 90, C 0, E1 0, E2 0, E3 0, E4 0 } C_DIS
LIN{ E6POS: X 749.3379, Y -16.9187, Z -110.0150, A 0, B 90, C 0, E1 0, E2 0, E3 0, E4 0 } C_DIS
LIN{ E6POS: X 748.3381, Y -16.8998, Z -110.0150, A 0, B 90, C 0, E1 0, E2 0, E3 0, E4 0 } C_DIS
LIN{ E6POS: X 747.3383, Y -16.8809, Z -110.0150, A 0, B 90, C 0, E1 0, E2 0, E3 0, E4 0 } C_DIS
LIN{ E6POS: X 746.3385, Y -16.8620, Z -110.0150, A 0, B 90, C 0, E1 0, E2 0, E3 0, E4 0 } C_DIS
LIN{ E6POS: X 745.3387, Y -16.8431, Z -110.0150, A 0, B 90, C 0, E1 0, E2 0, E3 0, E4 0 } C_DIS
LIN{ E6POS: X 744.5289, Y -16.8278, Z -110.0150, A 0, B 90, C 0, E1 0, E2 0, E3 0, E4 0 } C_DIS
LIN{ E6POS: X 743.5299, Y -16.8726, Z -110.0150, A 0, B 90, C 0, E1 0, E2 0, E3 0, E4 0 } C_DIS
LIN{ E6POS: X 742.5309, Y -16.9173, Z -110.0150, A 0, B 90, C 0, E1 0, E2 0, E3 0, E4 0 } C_DIS
LIN{ E6POS: X 741.7393, Y -16.9528, Z -110.0150, A 0, B 90, C 0, E1 0, E2 0, E3 0, E4 0 } C_DIS
LIN{ E6POS: X 740.7399, Y -16.9874, Z -110.0150, A 0, B 90, C 0, E1 0, E2 0, E3 0, E4 0 } C_DIS
LIN{ E6POS: X 739.7405, Y -17.0220, Z -110.0150, A 0, B 90, C 0, E1 0, E2 0, E3 0, E4 0 } C_DIS
LIN{ E6POS: X 738.7411, Y -17.0566, Z -110.0150, A 0, B 90, C 0, E1 0, E2 0, E3 0, E4 0 } C_DIS
LIN{ E6POS: X 737.8641, Y -17.0869, Z -110.0150, A 0, B 90, C 0, E1 0, E2 0, E3 0, E4 0 } C_DIS
LIN{ E6POS: X 736.8792, Y -17.2601, Z -110.0150, A 0, B 90, C 0, E1 0, E2 0, E3 0, E4 0 } C_DIS
LIN{ E6POS: X 736.1867, Y -17.3820, Z -110.0150, A 0, B 90, C 0, E1 0, E2 0, E3 0, E4 0 } C_DIS
LIN{ E6POS: X 735.1975, Y -17.5285, Z -110.0150, A 0, B 90, C 0, E1 0, E2 0, E3 0, E4 0 } C_DIS
LIN{ E6POS: X 734.2083, Y -17.6750, Z -110.0150, A 0, B 90, C 0, E1 0, E2 0, E3 0, E4 0 } C_DIS
LIN{ E6POS: X 733.8604, Y -17.7266, Z -110.0150, A 0, B 90, C 0, E1 0, E2 0, E3 0, E4 0 } C_DIS
LIN{ E6POS: X 733.2967, Y -18.1812, Z -110.0150, A 0, B 90, C 0, E1 0, E2 0, E3 0, E4 0 } C_DIS
LIN{ E6POS: X 732.5190, Y -18.7315, Z -110.0150, A 0, B 90, C 0, E1 0, E2 0, E3 0, E4 0 } C_DIS
LIN{ E6POS: X 733.2355, Y -19.4290, Z -110.0150, A 0, B 90, C 0, E1 0, E2 0, E3 0, E4 0 } C_DIS
LIN{ E6POS: X 733.2897, Y -19.4818, Z -110.0150, A 0, B 90, C 0, E1 0, E2 0, E3 0, E4 0 } C_DIS
LIN{ E6POS: X 733.8405, Y -20.0875, Z -110.0150, A 0, B 90, C 0, E1 0, E2 0, E3 0, E4 0 } C_DIS
LIN{ E6POS: X 734.7664, Y -20.4654, Z -110.0150, A 0, B 90, C 0, E1 0, E2 0, E3 0, E4 0 } C_DIS
LIN{ E6POS: X 735.6922, Y -20.8433, Z -110.0150, A 0, B 90, C 0, E1 0, E2 0, E3 0, E4 0 } C_DIS
LIN{ E6POS: X 736.1596, Y -21.0341, Z -110.0150, A 0, B 90, C 0, E1 0, E2 0, E3 0, E4 0 } C_DIS
LIN{ E6POS: X 737.0721, Y -21.4432, Z -110.0150, A 0, B 90, C 0, E1 0, E2 0, E3 0, E4 0 } C_DIS
LIN{ E6POS: X 737.8255, Y -21.7810, Z -110.0150, A 0, B 90, C 0, E1 0, E2 0, E3 0, E4 0 } C_DIS
LIN{ E6POS: X 738.7848, Y -22.0634, Z -110.0150, A 0, B 90, C 0, E1 0, E2 0, E3 0, E4 0 } C_DIS
LIN{ E6POS: X 739.7441, Y -22.3457, Z -110.0150, A 0, B 90, C 0, E1 0, E2 0, E3 0, E4 0 } C_DIS
LIN{ E6POS: X 740.7034, Y -22.6281, Z -110.0150, A 0, B 90, C 0, E1 0, E2 0, E3 0, E4 0 } C_DIS
LIN{ E6POS: X 741.6627, Y -22.9104, Z -110.0150, A 0, B 90, C 0, E1 0, E2 0, E3 0, E4 0 } C_DIS
LIN{ E6POS: X 741.6921, Y -22.9191, Z -110.0150, A 0, B 90, C 0, E1 0, E2 0, E3 0, E4 0 } C_DIS
LIN{ E6POS: X 742.6457, Y -23.2202, Z -110.0150, A 0, B 90, C 0, E1 0, E2 0, E3 0, E4 0 } C_DIS
LIN{ E6POS: X 743.5993, Y -23.5213, Z -110.0150, A 0, B 90, C 0, E1 0, E2 0, E3 0, E4 0 } C_DIS
LIN{ E6POS: X 744.4742, Y -23.7976, Z -110.0150, A 0, B 90, C 0, E1 0, E2 0, E3 0, E4 0 } C_DIS
LIN{ E6POS: X 745.4466, Y -24.0310, Z -110.0150, A 0, B 90, C 0, E1 0, E2 0, E3 0, E4 0 } C_DIS
LIN{ E6POS: X 746.4190, Y -24.2644, Z -110.0150, A 0, B 90, C 0, E1 0, E2 0, E3 0, E4 0 } C_DIS
LIN{ E6POS: X 747.3914, Y -24.4978, Z -110.0150, A 0, B 90, C 0, E1 0, E2 0, E3 0, E4 0 } C_DIS
LIN{ E6POS: X 748.3637, Y -24.7313, Z -110.0150, A 0, B 90, C 0, E1 0, E2 0, E3 0, E4 0 } C_DIS
LIN{ E6POS: X 749.2755, Y -24.9501, Z -110.0150, A 0, B 90, C 0, E1 0, E2 0, E3 0, E4 0 } C_DIS
LIN{ E6POS: X 750.2448, Y -25.1959, Z -110.0150, A 0, B 90, C 0, E1 0, E2 0, E3 0, E4 0 } C_DIS
LIN{ E6POS: X 751.2142, Y -25.4417, Z -110.0150, A 0, B 90, C 0, E1 0, E2 0, E3 0, E4 0 } C_DIS
LIN{ E6POS: X 752.1835, Y -25.6874, Z -110.0150, A 0, B 90, C 0, E1 0, E2 0, E3 0, E4 0 } C_DIS
LIN{ E6POS: X 752.7426, Y -25.8292, Z -110.0150, A 0, B 90, C 0, E1 0, E2 0, E3 0, E4 0 } C_DIS
LIN{ E6POS: X 753.7244, Y -26.0192, Z -110.0150, A 0, B 90, C 0, E1 0, E2 0, E3 0, E4 0 } C_DIS
LIN{ E6POS: X 754.7062, Y -26.2091, Z -110.0150, A 0, B 90, C 0, E1 0, E2 0, E3 0, E4 0 } C_DIS
LIN{ E6POS: X 755.6880, Y -26.3991, Z -110.0150, A 0, B 90, C 0, E1 0, E2 0, E3 0, E4 0 } C_DIS
LIN{ E6POS: X 756.6698, Y -26.5891, Z -110.0150, A 0, B 90, C 0, E1 0, E2 0, E3 0, E4 0 } C_DIS
LIN{ E6POS: X 757.6516, Y -26.7791, Z -110.0150, A 0, B 90, C 0, E1 0, E2 0, E3 0, E4 0 } C_DIS
LIN{ E6POS: X 757.8650, Y -26.8204, Z -110.0150, A 0, B 90, C 0, E1 0, E2 0, E3 0, E4 0 } C_DIS
LIN{ E6POS: X 758.8453, Y -27.0176, Z -110.0150, A 0, B 90, C 0, E1 0, E2 0, E3 0, E4 0 } C_DIS
LIN{ E6POS: X 759.8257, Y -27.2148, Z -110.0150, A 0, B 90, C 0, E1 0, E2 0, E3 0, E4 0 } C_DIS
LIN{ E6POS: X 760.8061, Y -27.4120, Z -110.0150, A 0, B 90, C 0, E1 0, E2 0, E3 0, E4 0 } C_DIS
LIN{ E6POS: X 761.5846, Y -27.5686, Z -110.0150, A 0, B 90, C 0, E1 0, E2 0, E3 0, E4 0 } C_DIS
LIN{ E6POS: X 762.5756, Y -27.7026, Z -110.0150, A 0, B 90, C 0, E1 0, E2 0, E3 0, E4 0 } C_DIS
LIN{ E6POS: X 763.5666, Y -27.8366, Z -110.0150, A 0, B 90, C 0, E1 0, E2 0, E3 0, E4 0 } C_DIS
LIN{ E6POS: X 764.5575, Y -27.9707, Z -110.0150, A 0, B 90, C 0, E1 0, E2 0, E3 0, E4 0 } C_DIS
LIN{ E6POS: X 765.5485, Y -28.1047, Z -110.0150, A 0, B 90, C 0, E1 0, E2 0, E3 0, E4 0 } C_DIS
LIN{ E6POS: X 766.4136, Y -28.2217, Z -110.0150, A 0, B 90, C 0, E1 0, E2 0, E3 0, E4 0 } C_DIS
LIN{ E6POS: X 767.4043, Y -28.3577, Z -110.0150, A 0, B 90, C 0, E1 0, E2 0, E3 0, E4 0 } C_DIS
LIN{ E6POS: X 768.3950, Y -28.4936, Z -110.0150, A 0, B 90, C 0, E1 0, E2 0, E3 0, E4 0 } C_DIS
LIN{ E6POS: X 769.3857, Y -28.6296, Z -110.0150, A 0, B 90, C 0, E1 0, E2 0, E3 0, E4 0 } C_DIS
LIN{ E6POS: X 769.9549, Y -28.7077, Z -110.0150, A 0, B 90, C 0, E1 0, E2 0, E3 0, E4 0 } C_DIS
LIN{ E6POS: X 770.9543, Y -28.7432, Z -110.0150, A 0, B 90, C 0, E1 0, E2 0, E3 0, E4 0 } C_DIS
LIN{ E6POS: X 771.9536, Y -28.7788, Z -110.0150, A 0, B 90, C 0, E1 0, E2 0, E3 0, E4 0 } C_DIS
LIN{ E6POS: X 772.9530, Y -28.8143, Z -110.0150, A 0, B 90, C 0, E1 0, E2 0, E3 0, E4 0 } C_DIS
LIN{ E6POS: X 773.8784, Y -28.8472, Z -110.0150, A 0, B 90, C 0, E1 0, E2 0, E3 0, E4 0 } C_DIS
LIN{ E6POS: X 774.8779, Y -28.8789, Z -110.0150, A 0, B 90, C 0, E1 0, E2 0, E3 0, E4 0 } C_DIS
LIN{ E6POS: X 775.8774, Y -28.9106, Z -110.0150, A 0, B 90, C 0, E1 0, E2 0, E3 0, E4 0 } C_DIS
LIN{ E6POS: X 776.8088, Y -28.9401, Z -110.0150, A 0, B 90, C 0, E1 0, E2 0, E3 0, E4 0 } C_DIS
LIN{ E6POS: X 777.7919, Y -29.1230, Z -110.0150, A 0, B 90, C 0, E1 0, E2 0, E3 0, E4 0 } C_DIS
LIN{ E6POS: X 778.7751, Y -29.3059, Z -110.0150, A 0, B 90, C 0, E1 0, E2 0, E3 0, E4 0 } C_DIS
LIN{ E6POS: X 779.7225, Y -29.4822, Z -110.0150, A 0, B 90, C 0, E1 0, E2 0, E3 0, E4 0 } C_DIS
LIN{ E6POS: X 780.7051, Y -29.6678, Z -110.0150, A 0, B 90, C 0, E1 0, E2 0, E3 0, E4 0 } C_DIS
LIN{ E6POS: X 781.6878, Y -29.8534, Z -110.0150, A 0, B 90, C 0, E1 0, E2 0, E3 0, E4 0 } C_DIS
LIN{ E6POS: X 781.9360, Y -29.9003, Z -110.0150, A 0, B 90, C 0, E1 0, E2 0, E3 0, E4 0 } C_DIS
LIN{ E6POS: X 782.6309, Y -30.6193, Z -110.0150, A 0, B 90, C 0, E1 0, E2 0, E3 0, E4 0 } C_DIS
LIN{ E6POS: X 783.3258, Y -31.3384, Z -110.0150, A 0, B 90, C 0, E1 0, E2 0, E3 0, E4 0 } C_DIS
LIN{ E6POS: X 783.7378, Y -31.7647, Z -110.0150, A 0, B 90, C 0, E1 0, E2 0, E3 0, E4 0 } C_DIS
LIN{ E6POS: X 784.4269, Y -32.4893, Z -110.0150, A 0, B 90, C 0, E1 0, E2 0, E3 0, E4 0 } C_DIS
LIN{ E6POS: X 785.1160, Y -33.2139, Z -110.0150, A 0, B 90, C 0, E1 0, E2 0, E3 0, E4 0 } C_DIS
LIN{ E6POS: X 785.1281, Y -33.2266, Z -110.0150, A 0, B 90, C 0, E1 0, E2 0, E3 0, E4 0 } C_DIS
LIN{ E6POS: X 785.2695, Y -34.2166, Z -110.0150, A 0, B 90, C 0, E1 0, E2 0, E3 0, E4 0 } C_DIS
LIN{ E6POS: X 785.4109, Y -35.2065, Z -110.0150, A 0, B 90, C 0, E1 0, E2 0, E3 0, E4 0 } C_DIS
LIN{ E6POS: X 785.5523, Y -36.1965, Z -110.0150, A 0, B 90, C 0, E1 0, E2 0, E3 0, E4 0 } C_DIS
LIN{ E6POS: X 785.6937, Y -37.1864, Z -110.0150, A 0, B 90, C 0, E1 0, E2 0, E3 0, E4 0 } C_DIS
LIN{ E6POS: X 785.7142, Y -37.3297, Z -110.0150, A 0, B 90, C 0, E1 0, E2 0, E3 0, E4 0 } C_DIS
LIN{ E6POS: X 785.8556, Y -38.3197, Z -110.0150, A 0, B 90, C 0, E1 0, E2 0, E3 0, E4 0 } C_DIS
LIN{ E6POS: X 785.9970, Y -39.3096, Z -110.0150, A 0, B 90, C 0, E1 0, E2 0, E3 0, E4 0 } C_DIS
LIN{ E6POS: X 786.1384, Y -40.2996, Z -110.0150, A 0, B 90, C 0, E1 0, E2 0, E3 0, E4 0 } C_DIS
LIN{ E6POS: X 786.1747, Y -40.5536, Z -110.0150, A 0, B 90, C 0, E1 0, E2 0, E3 0, E4 0 } C_DIS
LIN{ E6POS: X 786.0743, Y -41.5485, Z -110.0150, A 0, B 90, C 0, E1 0, E2 0, E3 0, E4 0 } C_DIS
LIN{ E6POS: X 785.9740, Y -42.5435, Z -110.0150, A 0, B 90, C 0, E1 0, E2 0, E3 0, E4 0 } C_DIS
LIN{ E6POS: X 785.8737, Y -43.5384, Z -110.0150, A 0, B 90, C 0, E1 0, E2 0, E3 0, E4 0 } C_DIS
LIN{ E6POS: X 785.7734, Y -44.5334, Z -110.0150, A 0, B 90, C 0, E1 0, E2 0, E3 0, E4 0 } C_DIS
LIN{ E6POS: X 785.6731, Y -45.5283, Z -110.0150, A 0, B 90, C 0, E1 0, E2 0, E3 0, E4 0 } C_DIS
LIN{ E6POS: X 785.5728, Y -46.5233, Z -110.0150, A 0, B 90, C 0, E1 0, E2 0, E3 0, E4 0 } C_DIS
LIN{ E6POS: X 785.4725, Y -47.5183, Z -110.0150, A 0, B 90, C 0, E1 0, E2 0, E3 0, E4 0 } C_DIS
LIN{ E6POS: X 785.4427, Y -47.8139, Z -110.0150, A 0, B 90, C 0, E1 0, E2 0, E3 0, E4 0 } C_DIS
LIN{ E6POS: X 785.3423, Y -48.8089, Z -110.0150, A 0, B 90, C 0, E1 0, E2 0, E3 0, E4 0 } C_DIS
LIN{ E6POS: X 785.2420, Y -49.8038, Z -110.0150, A 0, B 90, C 0, E1 0, E2 0, E3 0, E4 0 } C_DIS
LIN{ E6POS: X 785.1417, Y -50.7988, Z -110.0150, A 0, B 90, C 0, E1 0, E2 0, E3 0, E4 0 } C_DIS
LIN{ E6POS: X 785.0414, Y -51.7937, Z -110.0150, A 0, B 90, C 0, E1 0, E2 0, E3 0, E4 0 } C_DIS
LIN{ E6POS: X 784.9411, Y -52.7887, Z -110.0150, A 0, B 90, C 0, E1 0, E2 0, E3 0, E4 0 } C_DIS
LIN{ E6POS: X 784.8675, Y -53.5185, Z -110.0150, A 0, B 90, C 0, E1 0, E2 0, E3 0, E4 0 } C_DIS
LIN{ E6POS: X 784.6915, Y -54.5029, Z -110.0150, A 0, B 90, C 0, E1 0, E2 0, E3 0, E4 0 } C_DIS
LIN{ E6POS: X 784.5156, Y -55.4873, Z -110.0150, A 0, B 90, C 0, E1 0, E2 0, E3 0, E4 0 } C_DIS
LIN{ E6POS: X 784.3396, Y -56.4717, Z -110.0150, A 0, B 90, C 0, E1 0, E2 0, E3 0, E4 0 } C_DIS
LIN{ E6POS: X 784.1637, Y -57.4560, Z -110.0150, A 0, B 90, C 0, E1 0, E2 0, E3 0, E4 0 } C_DIS
LIN{ E6POS: X 783.9877, Y -58.4404, Z -110.0150, A 0, B 90, C 0, E1 0, E2 0, E3 0, E4 0 } C_DIS
LIN{ E6POS: X 783.8118, Y -59.4248, Z -110.0150, A 0, B 90, C 0, E1 0, E2 0, E3 0, E4 0 } C_DIS
LIN{ E6POS: X 783.6358, Y -60.4092, Z -110.0150, A 0, B 90, C 0, E1 0, E2 0, E3 0, E4 0 } C_DIS
LIN{ E6POS: X 783.4599, Y -61.3936, Z -110.0150, A 0, B 90, C 0, E1 0, E2 0, E3 0, E4 0 } C_DIS
LIN{ E6POS: X 783.2839, Y -62.3780, Z -110.0150, A 0, B 90, C 0, E1 0, E2 0, E3 0, E4 0 } C_DIS
LIN{ E6POS: X 783.1465, Y -63.1468, Z -110.0150, A 0, B 90, C 0, E1 0, E2 0, E3 0, E4 0 } C_DIS
LIN{ E6POS: X 782.9706, Y -64.1312, Z -110.0150, A 0, B 90, C 0, E1 0, E2 0, E3 0, E4 0 } C_DIS
LIN{ E6POS: X 782.7946, Y -65.1156, Z -110.0150, A 0, B 90, C 0, E1 0, E2 0, E3 0, E4 0 } C_DIS
LIN{ E6POS: X 782.6187, Y -66.0999, Z -110.0150, A 0, B 90, C 0, E1 0, E2 0, E3 0, E4 0 } C_DIS
LIN{ E6POS: X 782.4427, Y -67.0843, Z -110.0150, A 0, B 90, C 0, E1 0, E2 0, E3 0, E4 0 } C_DIS
LIN{ E6POS: X 782.2668, Y -68.0687, Z -110.0150, A 0, B 90, C 0, E1 0, E2 0, E3 0, E4 0 } C_DIS
LIN{ E6POS: X 782.0908, Y -69.0531, Z -110.0150, A 0, B 90, C 0, E1 0, E2 0, E3 0, E4 0 } C_DIS
LIN{ E6POS: X 781.9149, Y -70.0375, Z -110.0150, A 0, B 90, C 0, E1 0, E2 0, E3 0, E4 0 } C_DIS
LIN{ E6POS: X 781.7943, Y -70.7119, Z -110.0150, A 0, B 90, C 0, E1 0, E2 0, E3 0, E4 0 } C_DIS
LIN{ E6POS: X 781.5865, Y -71.6900, Z -110.0150, A 0, B 90, C 0, E1 0, E2 0, E3 0, E4 0 } C_DIS
LIN{ E6POS: X 781.3787, Y -72.6682, Z -110.0150, A 0, B 90, C 0, E1 0, E2 0, E3 0, E4 0 } C_DIS
LIN{ E6POS: X 781.1709, Y -73.6464, Z -110.0150, A 0, B 90, C 0, E1 0, E2 0, E3 0, E4 0 } C_DIS
LIN{ E6POS: X 780.9631, Y -74.6245, Z -110.0150, A 0, B 90, C 0, E1 0, E2 0, E3 0, E4 0 } C_DIS
LIN{ E6POS: X 780.7553, Y -75.6027, Z -110.0150, A 0, B 90, C 0, E1 0, E2 0, E3 0, E4 0 } C_DIS
LIN{ E6POS: X 780.5475, Y -76.5809, Z -110.0150, A 0, B 90, C 0, E1 0, E2 0, E3 0, E4 0 } C_DIS
LIN{ E6POS: X 780.3397, Y -77.5590, Z -110.0150, A 0, B 90, C 0, E1 0, E2 0, E3 0, E4 0 } C_DIS
LIN{ E6POS: X 780.1319, Y -78.5372, Z -110.0150, A 0, B 90, C 0, E1 0, E2 0, E3 0, E4 0 } C_DIS
LIN{ E6POS: X 779.9241, Y -79.5154, Z -110.0150, A 0, B 90, C 0, E1 0, E2 0, E3 0, E4 0 } C_DIS
LIN{ E6POS: X 779.7163, Y -80.4936, Z -110.0150, A 0, B 90, C 0, E1 0, E2 0, E3 0, E4 0 } C_DIS
LIN{ E6POS: X 779.5085, Y -81.4717, Z -110.0150, A 0, B 90, C 0, E1 0, E2 0, E3 0, E4 0 } C_DIS
LIN{ E6POS: X 779.4135, Y -81.9188, Z -110.0150, A 0, B 90, C 0, E1 0, E2 0, E3 0, E4 0 } C_DIS
LIN{ E6POS: X 779.2057, Y -82.8970, Z -110.0150, A 0, B 90, C 0, E1 0, E2 0, E3 0, E4 0 } C_DIS
LIN{ E6POS: X 778.9979, Y -83.8752, Z -110.0150, A 0, B 90, C 0, E1 0, E2 0, E3 0, E4 0 } C_DIS
LIN{ E6POS: X 778.7901, Y -84.8533, Z -110.0150, A 0, B 90, C 0, E1 0, E2 0, E3 0, E4 0 } C_DIS
LIN{ E6POS: X 778.5823, Y -85.8315, Z -110.0150, A 0, B 90, C 0, E1 0, E2 0, E3 0, E4 0 } C_DIS
LIN{ E6POS: X 778.3745, Y -86.8097, Z -110.0150, A 0, B 90, C 0, E1 0, E2 0, E3 0, E4 0 } C_DIS
LIN{ E6POS: X 778.1667, Y -87.7878, Z -110.0150, A 0, B 90, C 0, E1 0, E2 0, E3 0, E4 0 } C_DIS
LIN{ E6POS: X 777.9589, Y -88.7660, Z -110.0150, A 0, B 90, C 0, E1 0, E2 0, E3 0, E4 0 } C_DIS
LIN{ E6POS: X 777.7511, Y -89.7442, Z -110.0150, A 0, B 90, C 0, E1 0, E2 0, E3 0, E4 0 } C_DIS
LIN{ E6POS: X 777.5433, Y -90.7224, Z -110.0150, A 0, B 90, C 0, E1 0, E2 0, E3 0, E4 0 } C_DIS
LIN{ E6POS: X 777.5429, Y -90.7243, Z -110.0150, A 0, B 90, C 0, E1 0, E2 0, E3 0, E4 0 } C_DIS
LIN{ E6POS: X 777.3226, Y -91.6997, Z -110.0150, A 0, B 90, C 0, E1 0, E2 0, E3 0, E4 0 } C_DIS
LIN{ E6POS: X 777.1022, Y -92.6751, Z -110.0150, A 0, B 90, C 0, E1 0, E2 0, E3 0, E4 0 } C_DIS
LIN{ E6POS: X 776.8819, Y -93.6506, Z -110.0150, A 0, B 90, C 0, E1 0, E2 0, E3 0, E4 0 } C_DIS
LIN{ E6POS: X 776.6615, Y -94.6260, Z -110.0150, A 0, B 90, C 0, E1 0, E2 0, E3 0, E4 0 } C_DIS
LIN{ E6POS: X 776.4412, Y -95.6014, Z -110.0150, A 0, B 90, C 0, E1 0, E2 0, E3 0, E4 0 } C_DIS
LIN{ E6POS: X 776.2208, Y -96.5768, Z -110.0150, A 0, B 90, C 0, E1 0, E2 0, E3 0, E4 0 } C_DIS
LIN{ E6POS: X 776.0005, Y -97.5522, Z -110.0150, A 0, B 90, C 0, E1 0, E2 0, E3 0, E4 0 } C_DIS
LIN{ E6POS: X 775.7802, Y -98.5277, Z -110.0150, A 0, B 90, C 0, E1 0, E2 0, E3 0, E4 0 } C_DIS
LIN{ E6POS: X 775.5598, Y -99.5031, Z -110.0150, A 0, B 90, C 0, E1 0, E2 0, E3 0, E4 0 } C_DIS
LIN{ E6POS: X 775.3395, Y -100.4785, Z -110.0150, A 0, B 90, C 0, E1 0, E2 0, E3 0, E4 0 } C_DIS
LIN{ E6POS: X 775.1191, Y -101.4539, Z -110.0150, A 0, B 90, C 0, E1 0, E2 0, E3 0, E4 0 } C_DIS
LIN{ E6POS: X 774.8988, Y -102.4294, Z -110.0150, A 0, B 90, C 0, E1 0, E2 0, E3 0, E4 0 } C_DIS
LIN{ E6POS: X 774.8330, Y -102.7206, Z -110.0150, A 0, B 90, C 0, E1 0, E2 0, E3 0, E4 0 } C_DIS
LIN{ E6POS: X 774.6126, Y -103.6960, Z -110.0150, A 0, B 90, C 0, E1 0, E2 0, E3 0, E4 0 } C_DIS
LIN{ E6POS: X 774.3923, Y -104.6714, Z -110.0150, A 0, B 90, C 0, E1 0, E2 0, E3 0, E4 0 } C_DIS
LIN{ E6POS: X 774.1720, Y -105.6468, Z -110.0150, A 0, B 90, C 0, E1 0, E2 0, E3 0, E4 0 } C_DIS
LIN{ E6POS: X 773.9516, Y -106.6222, Z -110.0150, A 0, B 90, C 0, E1 0, E2 0, E3 0, E4 0 } C_DIS
LIN{ E6POS: X 773.7313, Y -107.5977, Z -110.0150, A 0, B 90, C 0, E1 0, E2 0, E3 0, E4 0 } C_DIS
LIN{ E6POS: X 773.5109, Y -108.5731, Z -110.0150, A 0, B 90, C 0, E1 0, E2 0, E3 0, E4 0 } C_DIS
LIN{ E6POS: X 773.2906, Y -109.5485, Z -110.0150, A 0, B 90, C 0, E1 0, E2 0, E3 0, E4 0 } C_DIS
LIN{ E6POS: X 773.0702, Y -110.5239, Z -110.0150, A 0, B 90, C 0, E1 0, E2 0, E3 0, E4 0 } C_DIS
LIN{ E6POS: X 772.8499, Y -111.4994, Z -110.0150, A 0, B 90, C 0, E1 0, E2 0, E3 0, E4 0 } C_DIS
LIN{ E6POS: X 772.7038, Y -112.1462, Z -110.0150, A 0, B 90, C 0, E1 0, E2 0, E3 0, E4 0 } C_DIS
LIN{ E6POS: X 772.0412, Y -111.3972, Z -110.0150, A 0, B 90, C 0, E1 0, E2 0, E3 0, E4 0 } C_DIS
LIN{ E6POS: X 771.3787, Y -110.6481, Z -110.0150, A 0, B 90, C 0, E1 0, E2 0, E3 0, E4 0 } C_DIS
LIN{ E6POS: X 771.2073, Y -110.4543, Z -110.0150, A 0, B 90, C 0, E1 0, E2 0, E3 0, E4 0 } C_DIS
LIN{ E6POS: X 770.5448, Y -109.7053, Z -110.0150, A 0, B 90, C 0, E1 0, E2 0, E3 0, E4 0 } C_DIS
LIN{ E6POS: X 770.0315, Y -109.1250, Z -110.0150, A 0, B 90, C 0, E1 0, E2 0, E3 0, E4 0 } C_DIS
LIN{ E6POS: X 769.2897, Y -108.4544, Z -110.0150, A 0, B 90, C 0, E1 0, E2 0, E3 0, E4 0 } C_DIS
LIN{ E6POS: X 768.5479, Y -107.7838, Z -110.0150, A 0, B 90, C 0, E1 0, E2 0, E3 0, E4 0 } C_DIS
LIN{ E6POS: X 768.0714, Y -107.3530, Z -110.0150, A 0, B 90, C 0, E1 0, E2 0, E3 0, E4 0 } C_DIS
LIN{ E6POS: X 767.3304, Y -106.6815, Z -110.0150, A 0, B 90, C 0, E1 0, E2 0, E3 0, E4 0 } C_DIS
LIN{ E6POS: X 766.5894, Y -106.0100, Z -110.0150, A 0, B 90, C 0, E1 0, E2 0, E3 0, E4 0 } C_DIS
LIN{ E6POS: X 766.5418, Y -105.9668, Z -110.0150, A 0, B 90, C 0, E1 0, E2 0, E3 0, E4 0 } C_DIS
LIN{ E6POS: X 765.7111, Y -105.4101, Z -110.0150, A 0, B 90, C 0, E1 0, E2 0, E3 0, E4 0 } C_DIS
LIN{ E6POS: X 764.8804, Y -104.8534, Z -110.0150, A 0, B 90, C 0, E1 0, E2 0, E3 0, E4 0 } C_DIS
LIN{ E6POS: X 764.3054, Y -104.4680, Z -110.0150, A 0, B 90, C 0, E1 0, E2 0, E3 0, E4 0 } C_DIS
LIN{ E6POS: X 763.4743, Y -103.9120, Z -110.0150, A 0, B 90, C 0, E1 0, E2 0, E3 0, E4 0 } C_DIS
LIN{ E6POS: X 762.6431, Y -103.3561, Z -110.0150, A 0, B 90, C 0, E1 0, E2 0, E3 0, E4 0 } C_DIS
LIN{ E6POS: X 761.8119, Y -102.8001, Z -110.0150, A 0, B 90, C 0, E1 0, E2 0, E3 0, E4 0 } C_DIS
LIN{ E6POS: X 761.4179, Y -102.5365, Z -110.0150, A 0, B 90, C 0, E1 0, E2 0, E3 0, E4 0 } C_DIS
LIN{ E6POS: X 760.5257, Y -102.0849, Z -110.0150, A 0, B 90, C 0, E1 0, E2 0, E3 0, E4 0 } C_DIS
LIN{ E6POS: X 759.6334, Y -101.6334, Z -110.0150, A 0, B 90, C 0, E1 0, E2 0, E3 0, E4 0 } C_DIS
LIN{ E6POS: X 758.7412, Y -101.1818, Z -110.0150, A 0, B 90, C 0, E1 0, E2 0, E3 0, E4 0 } C_DIS
LIN{ E6POS: X 758.1207, Y -100.8678, Z -110.0150, A 0, B 90, C 0, E1 0, E2 0, E3 0, E4 0 } C_DIS
LIN{ E6POS: X 757.2290, Y -100.4152, Z -110.0150, A 0, B 90, C 0, E1 0, E2 0, E3 0, E4 0 } C_DIS
LIN{ E6POS: X 756.3373, Y -99.9627, Z -110.0150, A 0, B 90, C 0, E1 0, E2 0, E3 0, E4 0 } C_DIS
LIN{ E6POS: X 755.4455, Y -99.5102, Z -110.0150, A 0, B 90, C 0, E1 0, E2 0, E3 0, E4 0 } C_DIS
LIN{ E6POS: X 754.5538, Y -99.0577, Z -110.0150, A 0, B 90, C 0, E1 0, E2 0, E3 0, E4 0 } C_DIS
LIN{ E6POS: X 753.8426, Y -98.6968, Z -110.0150, A 0, B 90, C 0, E1 0, E2 0, E3 0, E4 0 } C_DIS
LIN{ E6POS: X 752.9149, Y -98.3235, Z -110.0150, A 0, B 90, C 0, E1 0, E2 0, E3 0, E4 0 } C_DIS
LIN{ E6POS: X 751.9871, Y -97.9503, Z -110.0150, A 0, B 90, C 0, E1 0, E2 0, E3 0, E4 0 } C_DIS
LIN{ E6POS: X 751.0594, Y -97.5770, Z -110.0150, A 0, B 90, C 0, E1 0, E2 0, E3 0, E4 0 } C_DIS
LIN{ E6POS: X 750.1317, Y -97.2038, Z -110.0150, A 0, B 90, C 0, E1 0, E2 0, E3 0, E4 0 } C_DIS
LIN{ E6POS: X 749.2039, Y -96.8305, Z -110.0150, A 0, B 90, C 0, E1 0, E2 0, E3 0, E4 0 } C_DIS
LIN{ E6POS: X 749.1316, Y -96.8014, Z -110.0150, A 0, B 90, C 0, E1 0, E2 0, E3 0, E4 0 } C_DIS
LIN{ E6POS: X 748.2051, Y -96.4251, Z -110.0150, A 0, B 90, C 0, E1 0, E2 0, E3 0, E4 0 } C_DIS
LIN{ E6POS: X 747.2786, Y -96.0489, Z -110.0150, A 0, B 90, C 0, E1 0, E2 0, E3 0, E4 0 } C_DIS
LIN{ E6POS: X 746.3521, Y -95.6726, Z -110.0150, A 0, B 90, C 0, E1 0, E2 0, E3 0, E4 0 } C_DIS
LIN{ E6POS: X 745.4255, Y -95.2963, Z -110.0150, A 0, B 90, C 0, E1 0, E2 0, E3 0, E4 0 } C_DIS
LIN{ E6POS: X 744.4990, Y -94.9200, Z -110.0150, A 0, B 90, C 0, E1 0, E2 0, E3 0, E4 0 } C_DIS
LIN{ E6POS: X 743.5725, Y -94.5438, Z -110.0150, A 0, B 90, C 0, E1 0, E2 0, E3 0, E4 0 } C_DIS
LIN{ E6POS: X 742.9987, Y -94.3107, Z -110.0150, A 0, B 90, C 0, E1 0, E2 0, E3 0, E4 0 } C_DIS
LIN{ E6POS: X 742.0584, Y -93.9705, Z -110.0150, A 0, B 90, C 0, E1 0, E2 0, E3 0, E4 0 } C_DIS
LIN{ E6POS: X 741.1180, Y -93.6302, Z -110.0150, A 0, B 90, C 0, E1 0, E2 0, E3 0, E4 0 } C_DIS
LIN{ E6POS: X 740.1777, Y -93.2899, Z -110.0150, A 0, B 90, C 0, E1 0, E2 0, E3 0, E4 0 } C_DIS
LIN{ E6POS: X 739.2374, Y -92.9497, Z -110.0150, A 0, B 90, C 0, E1 0, E2 0, E3 0, E4 0 } C_DIS
LIN{ E6POS: X 738.2970, Y -92.6094, Z -110.0150, A 0, B 90, C 0, E1 0, E2 0, E3 0, E4 0 } C_DIS
LIN{ E6POS: X 737.6574, Y -92.3780, Z -110.0150, A 0, B 90, C 0, E1 0, E2 0, E3 0, E4 0 } C_DIS
LIN{ E6POS: X 736.7183, Y -92.0342, Z -110.0150, A 0, B 90, C 0, E1 0, E2 0, E3 0, E4 0 } C_DIS
LIN{ E6POS: X 735.7792, Y -91.6905, Z -110.0150, A 0, B 90, C 0, E1 0, E2 0, E3 0, E4 0 } C_DIS
LIN{ E6POS: X 734.8402, Y -91.3468, Z -110.0150, A 0, B 90, C 0, E1 0, E2 0, E3 0, E4 0 } C_DIS
LIN{ E6POS: X 733.9011, Y -91.0030, Z -110.0150, A 0, B 90, C 0, E1 0, E2 0, E3 0, E4 0 } C_DIS
LIN{ E6POS: X 732.9620, Y -90.6593, Z -110.0150, A 0, B 90, C 0, E1 0, E2 0, E3 0, E4 0 } C_DIS
LIN{ E6POS: X 732.0230, Y -90.3156, Z -110.0150, A 0, B 90, C 0, E1 0, E2 0, E3 0, E4 0 } C_DIS
LIN{ E6POS: X 731.0839, Y -89.9718, Z -110.0150, A 0, B 90, C 0, E1 0, E2 0, E3 0, E4 0 } C_DIS
LIN{ E6POS: X 730.6934, Y -89.8289, Z -110.0150, A 0, B 90, C 0, E1 0, E2 0, E3 0, E4 0 } C_DIS
LIN{ E6POS: X 729.7477, Y -89.5040, Z -110.0150, A 0, B 90, C 0, E1 0, E2 0, E3 0, E4 0 } C_DIS
LIN{ E6POS: X 728.8019, Y -89.1791, Z -110.0150, A 0, B 90, C 0, E1 0, E2 0, E3 0, E4 0 } C_DIS
LIN{ E6POS: X 727.8562, Y -88.8542, Z -110.0150, A 0, B 90, C 0, E1 0, E2 0, E3 0, E4 0 } C_DIS
LIN{ E6POS: X 726.9104, Y -88.5293, Z -110.0150, A 0, B 90, C 0, E1 0, E2 0, E3 0, E4 0 } C_DIS
LIN{ E6POS: X 725.9647, Y -88.2044, Z -110.0150, A 0, B 90, C 0, E1 0, E2 0, E3 0, E4 0 } C_DIS
LIN{ E6POS: X 725.5056, Y -88.0467, Z -110.0150, A 0, B 90, C 0, E1 0, E2 0, E3 0, E4 0 } C_DIS
LIN{ E6POS: X 724.5608, Y -87.7191, Z -110.0150, A 0, B 90, C 0, E1 0, E2 0, E3 0, E4 0 } C_DIS
LIN{ E6POS: X 723.6160, Y -87.3915, Z -110.0150, A 0, B 90, C 0, E1 0, E2 0, E3 0, E4 0 } C_DIS
LIN{ E6POS: X 722.6712, Y -87.0639, Z -110.0150, A 0, B 90, C 0, E1 0, E2 0, E3 0, E4 0 } C_DIS
LIN{ E6POS: X 721.7264, Y -86.7363, Z -110.0150, A 0, B 90, C 0, E1 0, E2 0, E3 0, E4 0 } C_DIS
LIN{ E6POS: X 720.7815, Y -86.4087, Z -110.0150, A 0, B 90, C 0, E1 0, E2 0, E3 0, E4 0 } C_DIS
LIN{ E6POS: X 719.8367, Y -86.0811, Z -110.0150, A 0, B 90, C 0, E1 0, E2 0, E3 0, E4 0 } C_DIS
LIN{ E6POS: X 718.8919, Y -85.7535, Z -110.0150, A 0, B 90, C 0, E1 0, E2 0, E3 0, E4 0 } C_DIS
LIN{ E6POS: X 718.7327, Y -85.6983, Z -110.0150, A 0, B 90, C 0, E1 0, E2 0, E3 0, E4 0 } C_DIS
LIN{ E6POS: X 717.7858, Y -85.3768, Z -110.0150, A 0, B 90, C 0, E1 0, E2 0, E3 0, E4 0 } C_DIS
LIN{ E6POS: X 716.8389, Y -85.0553, Z -110.0150, A 0, B 90, C 0, E1 0, E2 0, E3 0, E4 0 } C_DIS
LIN{ E6POS: X 715.8920, Y -84.7338, Z -110.0150, A 0, B 90, C 0, E1 0, E2 0, E3 0, E4 0 } C_DIS
LIN{ E6POS: X 714.9451, Y -84.4123, Z -110.0150, A 0, B 90, C 0, E1 0, E2 0, E3 0, E4 0 } C_DIS
LIN{ E6POS: X 714.4827, Y -84.2552, Z -110.0150, A 0, B 90, C 0, E1 0, E2 0, E3 0, E4 0 } C_DIS
LIN{ E6POS: X 713.5356, Y -83.9340, Z -110.0150, A 0, B 90, C 0, E1 0, E2 0, E3 0, E4 0 } C_DIS
LIN{ E6POS: X 712.5886, Y -83.6129, Z -110.0150, A 0, B 90, C 0, E1 0, E2 0, E3 0, E4 0 } C_DIS
LIN{ E6POS: X 711.6416, Y -83.2917, Z -110.0150, A 0, B 90, C 0, E1 0, E2 0, E3 0, E4 0 } C_DIS
LIN{ E6POS: X 710.6946, Y -82.9705, Z -110.0150, A 0, B 90, C 0, E1 0, E2 0, E3 0, E4 0 } C_DIS
LIN{ E6POS: X 709.7476, Y -82.6493, Z -110.0150, A 0, B 90, C 0, E1 0, E2 0, E3 0, E4 0 } C_DIS
LIN{ E6POS: X 708.9236, Y -82.3698, Z -110.0150, A 0, B 90, C 0, E1 0, E2 0, E3 0, E4 0 } C_DIS
LIN{ E6POS: X 707.9833, Y -82.0295, Z -110.0150, A 0, B 90, C 0, E1 0, E2 0, E3 0, E4 0 } C_DIS
LIN{ E6POS: X 707.0430, Y -81.6892, Z -110.0150, A 0, B 90, C 0, E1 0, E2 0, E3 0, E4 0 } C_DIS
LIN{ E6POS: X 706.3946, Y -81.4545, Z -110.0150, A 0, B 90, C 0, E1 0, E2 0, E3 0, E4 0 } C_DIS
LIN{ E6POS: X 705.4508, Y -81.1241, Z -110.0150, A 0, B 90, C 0, E1 0, E2 0, E3 0, E4 0 } C_DIS
LIN{ E6POS: X 704.5070, Y -80.7936, Z -110.0150, A 0, B 90, C 0, E1 0, E2 0, E3 0, E4 0 } C_DIS
LIN{ E6POS: X 703.5631, Y -80.4632, Z -110.0150, A 0, B 90, C 0, E1 0, E2 0, E3 0, E4 0 } C_DIS
LIN{ E6POS: X 703.0730, Y -80.2916, Z -110.0150, A 0, B 90, C 0, E1 0, E2 0, E3 0, E4 0 } C_DIS
LIN{ E6POS: X 702.1509, Y -79.9046, Z -110.0150, A 0, B 90, C 0, E1 0, E2 0, E3 0, E4 0 } C_DIS
LIN{ E6POS: X 701.8348, Y -79.7720, Z -110.0150, A 0, B 90, C 0, E1 0, E2 0, E3 0, E4 0 } C_DIS
LIN{ E6POS: X 700.8993, Y -79.4186, Z -110.0150, A 0, B 90, C 0, E1 0, E2 0, E3 0, E4 0 } C_DIS
LIN{ E6POS: X 700.1905, Y -79.1509, Z -110.0150, A 0, B 90, C 0, E1 0, E2 0, E3 0, E4 0 } C_DIS
LIN{ E6POS: X 699.8491, Y -78.8125, Z -110.0150, A 0, B 90, C 0, E1 0, E2 0, E3 0, E4 0 } C_DIS
LIN{ E6POS: X 699.3465, Y -78.5002, Z -110.0150, A 0, B 90, C 0, E1 0, E2 0, E3 0, E4 0 } C_DIS
LIN{ E6POS: X 699.5034, Y -77.7303, Z -110.0150, A 0, B 90, C 0, E1 0, E2 0, E3 0, E4 0 } C_DIS
LIN{ E6POS: X 699.6652, Y -77.0692, Z -110.0150, A 0, B 90, C 0, E1 0, E2 0, E3 0, E4 0 } C_DIS
LIN{ E6POS: X 699.8146, Y -76.3203, Z -110.0150, A 0, B 90, C 0, E1 0, E2 0, E3 0, E4 0 } C_DIS
LIN{ E6POS: X 699.9609, Y -75.7015, Z -110.0150, A 0, B 90, C 0, E1 0, E2 0, E3 0, E4 0 } C_DIS
LIN{ E6POS: X 700.1186, Y -74.9430, Z -110.0150, A 0, B 90, C 0, E1 0, E2 0, E3 0, E4 0 } C_DIS
LIN{ E6POS: X 700.2681, Y -74.3266, Z -110.0150, A 0, B 90, C 0, E1 0, E2 0, E3 0, E4 0 } C_DIS
LIN{ E6POS: X 700.4372, Y -73.5523, Z -110.0150, A 0, B 90, C 0, E1 0, E2 0, E3 0, E4 0 } C_DIS
LIN{ E6POS: X 700.5918, Y -72.9399, Z -110.0150, A 0, B 90, C 0, E1 0, E2 0, E3 0, E4 0 } C_DIS
LIN{ E6POS: X 700.7766, Y -72.1455, Z -110.0150, A 0, B 90, C 0, E1 0, E2 0, E3 0, E4 0 } C_DIS
LIN{ E6POS: X 700.9378, Y -71.5369, Z -110.0150, A 0, B 90, C 0, E1 0, E2 0, E3 0, E4 0 } C_DIS
LIN{ E6POS: X 701.1321, Y -70.7240, Z -110.0150, A 0, B 90, C 0, E1 0, E2 0, E3 0, E4 0 } C_DIS
LIN{ E6POS: X 701.2967, Y -70.1133, Z -110.0150, A 0, B 90, C 0, E1 0, E2 0, E3 0, E4 0 } C_DIS
LIN{ E6POS: X 701.4935, Y -69.2825, Z -110.0150, A 0, B 90, C 0, E1 0, E2 0, E3 0, E4 0 } C_DIS
LIN{ E6POS: X 701.6578, Y -68.6630, Z -110.0150, A 0, B 90, C 0, E1 0, E2 0, E3 0, E4 0 } C_DIS
LIN{ E6POS: X 701.8507, Y -67.8171, Z -110.0150, A 0, B 90, C 0, E1 0, E2 0, E3 0, E4 0 } C_DIS
LIN{ E6POS: X 702.0112, Y -67.1818, Z -110.0150, A 0, B 90, C 0, E1 0, E2 0, E3 0, E4 0 } C_DIS
LIN{ E6POS: X 702.1931, Y -66.3207, Z -110.0150, A 0, B 90, C 0, E1 0, E2 0, E3 0, E4 0 } C_DIS
LIN{ E6POS: X 702.3467, Y -65.6626, Z -110.0150, A 0, B 90, C 0, E1 0, E2 0, E3 0, E4 0 } C_DIS
LIN{ E6POS: X 702.5171, Y -64.8033, Z -110.0150, A 0, B 90, C 0, E1 0, E2 0, E3 0, E4 0 } C_DIS
LIN{ E6POS: X 702.6628, Y -64.1386, Z -110.0150, A 0, B 90, C 0, E1 0, E2 0, E3 0, E4 0 } C_DIS
LIN{ E6POS: X 702.8200, Y -63.2960, Z -110.0150, A 0, B 90, C 0, E1 0, E2 0, E3 0, E4 0 } C_DIS
LIN{ E6POS: X 702.9576, Y -62.6402, Z -110.0150, A 0, B 90, C 0, E1 0, E2 0, E3 0, E4 0 } C_DIS
LIN{ E6POS: X 703.1002, Y -61.8315, Z -110.0150, A 0, B 90, C 0, E1 0, E2 0, E3 0, E4 0 } C_DIS
LIN{ E6POS: X 703.2293, Y -61.2009, Z -110.0150, A 0, B 90, C 0, E1 0, E2 0, E3 0, E4 0 } C_DIS
LIN{ E6POS: X 703.3561, Y -60.4414, Z -110.0150, A 0, B 90, C 0, E1 0, E2 0, E3 0, E4 0 } C_DIS
LIN{ E6POS: X 703.4764, Y -59.8511, Z -110.0150, A 0, B 90, C 0, E1 0, E2 0, E3 0, E4 0 } C_DIS
LIN{ E6POS: X 703.5927, Y -59.1162, Z -110.0150, A 0, B 90, C 0, E1 0, E2 0, E3 0, E4 0 } C_DIS
LIN{ E6POS: X 703.7060, Y -58.5470, Z -110.0150, A 0, B 90, C 0, E1 0, E2 0, E3 0, E4 0 } C_DIS
LIN{ E6POS: X 703.8169, Y -57.8122, Z -110.0150, A 0, B 90, C 0, E1 0, E2 0, E3 0, E4 0 } C_DIS
LIN{ E6POS: X 703.9265, Y -57.2428, Z -110.0150, A 0, B 90, C 0, E1 0, E2 0, E3 0, E4 0 } C_DIS
LIN{ E6POS: X 704.0379, Y -56.4837, Z -110.0150, A 0, B 90, C 0, E1 0, E2 0, E3 0, E4 0 } C_DIS
LIN{ E6POS: X 704.1460, Y -55.8946, Z -110.0150, A 0, B 90, C 0, E1 0, E2 0, E3 0, E4 0 } C_DIS
LIN{ E6POS: X 704.2627, Y -55.0859, Z -110.0150, A 0, B 90, C 0, E1 0, E2 0, E3 0, E4 0 } C_DIS
LIN{ E6POS: X 704.3714, Y -54.4558, Z -110.0150, A 0, B 90, C 0, E1 0, E2 0, E3 0, E4 0 } C_DIS
LIN{ E6POS: X 704.4891, Y -53.6230, Z -110.0150, A 0, B 90, C 0, E1 0, E2 0, E3 0, E4 0 } C_DIS
LIN{ E6POS: X 704.5966, Y -52.9729, Z -110.0150, A 0, B 90, C 0, E1 0, E2 0, E3 0, E4 0 } C_DIS
LIN{ E6POS: X 704.7100, Y -52.1405, Z -110.0150, A 0, B 90, C 0, E1 0, E2 0, E3 0, E4 0 } C_DIS
LIN{ E6POS: X 704.8142, Y -51.4907, Z -110.0150, A 0, B 90, C 0, E1 0, E2 0, E3 0, E4 0 } C_DIS
LIN{ E6POS: X 704.9136, Y -50.8609, Z -110.0150, A 0, B 90, C 0, E1 0, E2 0, E3 0, E4 0 } C_DIS
LIN{ E6POS: X 705.0185, Y -50.0532, Z -110.0150, A 0, B 90, C 0, E1 0, E2 0, E3 0, E4 0 } C_DIS
LIN{ E6POS: X 705.1110, Y -49.4647, Z -110.0150, A 0, B 90, C 0, E1 0, E2 0, E3 0, E4 0 } C_DIS
LIN{ E6POS: X 705.2027, Y -48.7064, Z -110.0150, A 0, B 90, C 0, E1 0, E2 0, E3 0, E4 0 } C_DIS
LIN{ E6POS: X 705.2888, Y -48.1607, Z -110.0150, A 0, B 90, C 0, E1 0, E2 0, E3 0, E4 0 } C_DIS
LIN{ E6POS: X 705.3684, Y -47.4638, Z -110.0150, A 0, B 90, C 0, E1 0, E2 0, E3 0, E4 0 } C_DIS
LIN{ E6POS: X 705.4887, Y -46.4711, Z -110.0150, A 0, B 90, C 0, E1 0, E2 0, E3 0, E4 0 } C_DIS
LIN{ E6POS: X 705.5836, Y -45.6882, Z -110.0150, A 0, B 90, C 0, E1 0, E2 0, E3 0, E4 0 } C_DIS
LIN{ E6POS: X 705.6635, Y -45.1891, Z -110.0150, A 0, B 90, C 0, E1 0, E2 0, E3 0, E4 0 } C_DIS
LIN{ E6POS: X 705.8310, Y -44.2032, Z -110.0150, A 0, B 90, C 0, E1 0, E2 0, E3 0, E4 0 } C_DIS
LIN{ E6POS: X 705.8399, Y -44.1503, Z -110.0150, A 0, B 90, C 0, E1 0, E2 0, E3 0, E4 0 } C_DIS
LIN{ E6POS: X 706.0029, Y -43.1636, Z -110.0150, A 0, B 90, C 0, E1 0, E2 0, E3 0, E4 0 } C_DIS
LIN{ E6POS: X 706.0079, Y -43.1331, Z -110.0150, A 0, B 90, C 0, E1 0, E2 0, E3 0, E4 0 } C_DIS
LIN{ E6POS: X 706.1320, Y -42.1408, Z -110.0150, A 0, B 90, C 0, E1 0, E2 0, E3 0, E4 0 } C_DIS
LIN{ E6POS: X 706.2163, Y -41.4659, Z -110.0150, A 0, B 90, C 0, E1 0, E2 0, E3 0, E4 0 } C_DIS
LIN{ E6POS: X 706.2877, Y -40.9582, Z -110.0150, A 0, B 90, C 0, E1 0, E2 0, E3 0, E4 0 } C_DIS
LIN{ E6POS: X 706.3581, Y -40.3009, Z -110.0150, A 0, B 90, C 0, E1 0, E2 0, E3 0, E4 0 } C_DIS
LIN{ E6POS: X 706.4301, Y -39.7440, Z -110.0150, A 0, B 90, C 0, E1 0, E2 0, E3 0, E4 0 } C_DIS
LIN{ E6POS: X 706.4998, Y -39.0381, Z -110.0150, A 0, B 90, C 0, E1 0, E2 0, E3 0, E4 0 } C_DIS
LIN{ E6POS: X 706.5709, Y -38.4557, Z -110.0150, A 0, B 90, C 0, E1 0, E2 0, E3 0, E4 0 } C_DIS
LIN{ E6POS: X 706.6352, Y -37.7342, Z -110.0150, A 0, B 90, C 0, E1 0, E2 0, E3 0, E4 0 } C_DIS
LIN{ E6POS: X 706.7027, Y -37.1512, Z -110.0150, A 0, B 90, C 0, E1 0, E2 0, E3 0, E4 0 } C_DIS
LIN{ E6POS: X 706.7570, Y -36.4458, Z -110.0150, A 0, B 90, C 0, E1 0, E2 0, E3 0, E4 0 } C_DIS
LIN{ E6POS: X 706.8183, Y -35.8855, Z -110.0150, A 0, B 90, C 0, E1 0, E2 0, E3 0, E4 0 } C_DIS
LIN{ E6POS: X 706.8664, Y -35.1799, Z -110.0150, A 0, B 90, C 0, E1 0, E2 0, E3 0, E4 0 } C_DIS
LIN{ E6POS: X 706.9234, Y -34.6278, Z -110.0150, A 0, B 90, C 0, E1 0, E2 0, E3 0, E4 0 } C_DIS
LIN{ E6POS: X 706.9697, Y -33.9065, Z -110.0150, A 0, B 90, C 0, E1 0, E2 0, E3 0, E4 0 } C_DIS
LIN{ E6POS: X 707.0253, Y -33.3458, Z -110.0150, A 0, B 90, C 0, E1 0, E2 0, E3 0, E4 0 } C_DIS
LIN{ E6POS: X 707.0736, Y -32.5919, Z -110.0150, A 0, B 90, C 0, E1 0, E2 0, E3 0, E4 0 } C_DIS
LIN{ E6POS: X 707.1287, Y -32.0073, Z -110.0150, A 0, B 90, C 0, E1 0, E2 0, E3 0, E4 0 } C_DIS
LIN{ E6POS: X 707.1822, Y -31.2044, Z -110.0150, A 0, B 90, C 0, E1 0, E2 0, E3 0, E4 0 } C_DIS
LIN{ E6POS: X 707.2393, Y -30.5797, Z -110.0150, A 0, B 90, C 0, E1 0, E2 0, E3 0, E4 0 } C_DIS
LIN{ E6POS: X 707.2948, Y -29.7530, Z -110.0150, A 0, B 90, C 0, E1 0, E2 0, E3 0, E4 0 } C_DIS
LIN{ E6POS: X 707.3520, Y -29.1086, Z -110.0150, A 0, B 90, C 0, E1 0, E2 0, E3 0, E4 0 } C_DIS
LIN{ E6POS: X 707.4049, Y -28.2816, Z -110.0150, A 0, B 90, C 0, E1 0, E2 0, E3 0, E4 0 } C_DIS
LIN{ E6POS: X 707.4603, Y -27.6376, Z -110.0150, A 0, B 90, C 0, E1 0, E2 0, E3 0, E4 0 } C_DIS
LIN{ E6POS: X 707.5065, Y -26.8365, Z -110.0150, A 0, B 90, C 0, E1 0, E2 0, E3 0, E4 0 } C_DIS
LIN{ E6POS: X 707.5580, Y -26.2128, Z -110.0150, A 0, B 90, C 0, E1 0, E2 0, E3 0, E4 0 } C_DIS
LIN{ E6POS: X 707.5936, Y -25.4613, Z -110.0150, A 0, B 90, C 0, E1 0, E2 0, E3 0, E4 0 } C_DIS
LIN{ E6POS: X 707.6395, Y -24.8784, Z -110.0150, A 0, B 90, C 0, E1 0, E2 0, E3 0, E4 0 } C_DIS
LIN{ E6POS: X 707.6683, Y -24.1557, Z -110.0150, A 0, B 90, C 0, E1 0, E2 0, E3 0, E4 0 } C_DIS
LIN{ E6POS: X 707.7097, Y -23.5983, Z -110.0150, A 0, B 90, C 0, E1 0, E2 0, E3 0, E4 0 } C_DIS
LIN{ E6POS: X 707.7353, Y -22.8815, Z -110.0150, A 0, B 90, C 0, E1 0, E2 0, E3 0, E4 0 } C_DIS
LIN{ E6POS: X 707.7735, Y -22.3332, Z -110.0150, A 0, B 90, C 0, E1 0, E2 0, E3 0, E4 0 } C_DIS
LIN{ E6POS: X 707.7998, Y -21.6016, Z -110.0150, A 0, B 90, C 0, E1 0, E2 0, E3 0, E4 0 } C_DIS
LIN{ E6POS: X 707.8365, Y -21.0482, Z -110.0150, A 0, B 90, C 0, E1 0, E2 0, E3 0, E4 0 } C_DIS
LIN{ E6POS: X 707.8665, Y -20.2793, Z -110.0150, A 0, B 90, C 0, E1 0, E2 0, E3 0, E4 0 } C_DIS
LIN{ E6POS: X 707.9030, Y -19.7043, Z -110.0150, A 0, B 90, C 0, E1 0, E2 0, E3 0, E4 0 } C_DIS
LIN{ E6POS: X 707.9360, Y -18.9073, Z -110.0150, A 0, B 90, C 0, E1 0, E2 0, E3 0, E4 0 } C_DIS
LIN{ E6POS: X 707.9719, Y -18.3166, Z -110.0150, A 0, B 90, C 0, E1 0, E2 0, E3 0, E4 0 } C_DIS
LIN{ E6POS: X 708.0075, Y -17.5017, Z -110.0150, A 0, B 90, C 0, E1 0, E2 0, E3 0, E4 0 } C_DIS
LIN{ E6POS: X 708.0437, Y -16.9002, Z -110.0150, A 0, B 90, C 0, E1 0, E2 0, E3 0, E4 0 } C_DIS
LIN{ E6POS: X 708.0847, Y -15.9010, Z -110.0150, A 0, B 90, C 0, E1 0, E2 0, E3 0, E4 0 } C_DIS
LIN{ E6POS: X 708.0896, Y -15.7805, Z -110.0150, A 0, B 90, C 0, E1 0, E2 0, E3 0, E4 0 } C_DIS
LIN{ E6POS: X 708.1464, Y -14.8781, Z -110.0150, A 0, B 90, C 0, E1 0, E2 0, E3 0, E4 0 } C_DIS
LIN{ E6POS: X 708.1621, Y -13.8782, Z -110.0150, A 0, B 90, C 0, E1 0, E2 0, E3 0, E4 0 } C_DIS
LIN{ E6POS: X 708.1665, Y -13.5944, Z -110.0150, A 0, B 90, C 0, E1 0, E2 0, E3 0, E4 0 } C_DIS
LIN{ E6POS: X 708.2231, Y -12.5960, Z -110.0150, A 0, B 90, C 0, E1 0, E2 0, E3 0, E4 0 } C_DIS
LIN{ E6POS: X 708.2272, Y -12.5239, Z -110.0150, A 0, B 90, C 0, E1 0, E2 0, E3 0, E4 0 } C_DIS
LIN{ E6POS: X 708.2360, Y -11.8560, Z -110.0150, A 0, B 90, C 0, E1 0, E2 0, E3 0, E4 0 } C_DIS
LIN{ E6POS: X 708.2618, Y -11.3368, Z -110.0150, A 0, B 90, C 0, E1 0, E2 0, E3 0, E4 0 } C_DIS
LIN{ E6POS: X 708.2748, Y -10.5934, Z -110.0150, A 0, B 90, C 0, E1 0, E2 0, E3 0, E4 0 } C_DIS
LIN{ E6POS: X 708.3025, Y -10.0166, Z -110.0150, A 0, B 90, C 0, E1 0, E2 0, E3 0, E4 0 } C_DIS
LIN{ E6POS: X 708.3212, Y -9.2244, Z -110.0150, A 0, B 90, C 0, E1 0, E2 0, E3 0, E4 0 } C_DIS
LIN{ E6POS: X 708.3503, Y -8.6087, Z -110.0150, A 0, B 90, C 0, E1 0, E2 0, E3 0, E4 0 } C_DIS
LIN{ E6POS: X 708.3702, Y -7.7930, Z -110.0150, A 0, B 90, C 0, E1 0, E2 0, E3 0, E4 0 } C_DIS
LIN{ E6POS: X 708.3996, Y -7.1582, Z -110.0150, A 0, B 90, C 0, E1 0, E2 0, E3 0, E4 0 } C_DIS
LIN{ E6POS: X 708.4188, Y -6.3434, Z -110.0150, A 0, B 90, C 0, E1 0, E2 0, E3 0, E4 0 } C_DIS
LIN{ E6POS: X 708.4468, Y -5.7095, Z -110.0150, A 0, B 90, C 0, E1 0, E2 0, E3 0, E4 0 } C_DIS
LIN{ E6POS: X 708.4615, Y -4.9201, Z -110.0150, A 0, B 90, C 0, E1 0, E2 0, E3 0, E4 0 } C_DIS
LIN{ E6POS: X 708.4880, Y -4.3064, Z -110.0150, A 0, B 90, C 0, E1 0, E2 0, E3 0, E4 0 } C_DIS
LIN{ E6POS: X 708.4957, Y -3.5671, Z -110.0150, A 0, B 90, C 0, E1 0, E2 0, E3 0, E4 0 } C_DIS
LIN{ E6POS: X 708.5193, Y -2.9936, Z -110.0150, A 0, B 90, C 0, E1 0, E2 0, E3 0, E4 0 } C_DIS
LIN{ E6POS: X 708.5222, Y -2.2809, Z -110.0150, A 0, B 90, C 0, E1 0, E2 0, E3 0, E4 0 } C_DIS
LIN{ E6POS: X 708.5439, Y -1.7278, Z -110.0150, A 0, B 90, C 0, E1 0, E2 0, E3 0, E4 0 } C_DIS
LIN{ E6POS: X 708.5457, Y -1.0153, Z -110.0150, A 0, B 90, C 0, E1 0, E2 0, E3 0, E4 0 } C_DIS
LIN{ E6POS: X 708.5664, Y -0.4628, Z -110.0150, A 0, B 90, C 0, E1 0, E2 0, E3 0, E4 0 } C_DIS
LIN{ E6POS: X 708.5706, Y 0.2734, Z -110.0150, A 0, B 90, C 0, E1 0, E2 0, E3 0, E4 0 } C_DIS
LIN{ E6POS: X 708.5915, Y 0.8441, Z -110.0150, A 0, B 90, C 0, E1 0, E2 0, E3 0, E4 0 } C_DIS
LIN{ E6POS: X 708.6011, Y 1.6281, Z -110.0150, A 0, B 90, C 0, E1 0, E2 0, E3 0, E4 0 } C_DIS
LIN{ E6POS: X 708.6229, Y 2.2378, Z -110.0150, A 0, B 90, C 0, E1 0, E2 0, E3 0, E4 0 } C_DIS
LIN{ E6POS: X 708.6351, Y 3.0461, Z -110.0150, A 0, B 90, C 0, E1 0, E2 0, E3 0, E4 0 } C_DIS
LIN{ E6POS: X 708.6579, Y 3.6743, Z -110.0150, A 0, B 90, C 0, E1 0, E2 0, E3 0, E4 0 } C_DIS
LIN{ E6POS: X 708.6693, Y 4.4816, Z -110.0150, A 0, B 90, C 0, E1 0, E2 0, E3 0, E4 0 } C_DIS
LIN{ E6POS: X 708.6911, Y 5.1092, Z -110.0150, A 0, B 90, C 0, E1 0, E2 0, E3 0, E4 0 } C_DIS
LIN{ E6POS: X 708.6994, Y 5.8901, Z -110.0150, A 0, B 90, C 0, E1 0, E2 0, E3 0, E4 0 } C_DIS
LIN{ E6POS: X 708.7201, Y 6.4974, Z -110.0150, A 0, B 90, C 0, E1 0, E2 0, E3 0, E4 0 } C_DIS
LIN{ E6POS: X 708.7220, Y 7.2286, Z -110.0150, A 0, B 90, C 0, E1 0, E2 0, E3 0, E4 0 } C_DIS
LIN{ E6POS: X 708.7412, Y 7.7961, Z -110.0150, A 0, B 90, C 0, E1 0, E2 0, E3 0, E4 0 } C_DIS
LIN{ E6POS: X 708.7395, Y 8.5010, Z -110.0150, A 0, B 90, C 0, E1 0, E2 0, E3 0, E4 0 } C_DIS
LIN{ E6POS: X 708.7571, Y 9.0480, Z -110.0150, A 0, B 90, C 0, E1 0, E2 0, E3 0, E4 0 } C_DIS
LIN{ E6POS: X 708.7556, Y 9.7517, Z -110.0150, A 0, B 90, C 0, E1 0, E2 0, E3 0, E4 0 } C_DIS
LIN{ E6POS: X 708.7734, Y 10.2978, Z -110.0150, A 0, B 90, C 0, E1 0, E2 0, E3 0, E4 0 } C_DIS
LIN{ E6POS: X 708.7743, Y 11.0251, Z -110.0150, A 0, B 90, C 0, E1 0, E2 0, E3 0, E4 0 } C_DIS
LIN{ E6POS: X 708.7922, Y 11.5894, Z -110.0150, A 0, B 90, C 0, E1 0, E2 0, E3 0, E4 0 } C_DIS
LIN{ E6POS: X 708.7997, Y 12.3648, Z -110.0150, A 0, B 90, C 0, E1 0, E2 0, E3 0, E4 0 } C_DIS
LIN{ E6POS: X 708.8196, Y 12.9674, Z -110.0150, A 0, B 90, C 0, E1 0, E2 0, E3 0, E4 0 } C_DIS
LIN{ E6POS: X 708.8299, Y 13.7663, Z -110.0150, A 0, B 90, C 0, E1 0, E2 0, E3 0, E4 0 } C_DIS
LIN{ E6POS: X 708.8503, Y 14.3870, Z -110.0150, A 0, B 90, C 0, E1 0, E2 0, E3 0, E4 0 } C_DIS
LIN{ E6POS: X 708.8610, Y 15.1852, Z -110.0150, A 0, B 90, C 0, E1 0, E2 0, E3 0, E4 0 } C_DIS
LIN{ E6POS: X 708.8817, Y 15.8054, Z -110.0150, A 0, B 90, C 0, E1 0, E2 0, E3 0, E4 0 } C_DIS
LIN{ E6POS: X 708.8893, Y 16.5772, Z -110.0150, A 0, B 90, C 0, E1 0, E2 0, E3 0, E4 0 } C_DIS
LIN{ E6POS: X 708.9094, Y 17.1774, Z -110.0150, A 0, B 90, C 0, E1 0, E2 0, E3 0, E4 0 } C_DIS
LIN{ E6POS: X 708.9114, Y 17.8986, Z -110.0150, A 0, B 90, C 0, E1 0, E2 0, E3 0, E4 0 } C_DIS
LIN{ E6POS: X 708.9304, Y 18.4589, Z -110.0150, A 0, B 90, C 0, E1 0, E2 0, E3 0, E4 0 } C_DIS
LIN{ E6POS: X 708.9299, Y 19.1541, Z -110.0150, A 0, B 90, C 0, E1 0, E2 0, E3 0, E4 0 } C_DIS
LIN{ E6POS: X 708.9478, Y 19.6942, Z -110.0150, A 0, B 90, C 0, E1 0, E2 0, E3 0, E4 0 } C_DIS
LIN{ E6POS: X 708.9481, Y 20.3886, Z -110.0150, A 0, B 90, C 0, E1 0, E2 0, E3 0, E4 0 } C_DIS
LIN{ E6POS: X 708.9666, Y 20.9275, Z -110.0150, A 0, B 90, C 0, E1 0, E2 0, E3 0, E4 0 } C_DIS
LIN{ E6POS: X 708.9706, Y 21.6446, Z -110.0150, A 0, B 90, C 0, E1 0, E2 0, E3 0, E4 0 } C_DIS
LIN{ E6POS: X 708.9909, Y 22.2018, Z -110.0150, A 0, B 90, C 0, E1 0, E2 0, E3 0, E4 0 } C_DIS
LIN{ E6POS: X 709.0021, Y 22.9672, Z -110.0150, A 0, B 90, C 0, E1 0, E2 0, E3 0, E4 0 } C_DIS
LIN{ E6POS: X 709.0240, Y 23.5614, Z -110.0150, A 0, B 90, C 0, E1 0, E2 0, E3 0, E4 0 } C_DIS
LIN{ E6POS: X 709.0398, Y 24.3202, Z -110.0150, A 0, B 90, C 0, E1 0, E2 0, E3 0, E4 0 } C_DIS
LIN{ E6POS: X 709.0645, Y 24.9171, Z -110.0150, A 0, B 90, C 0, E1 0, E2 0, E3 0, E4 0 } C_DIS
LIN{ E6POS: X 709.0840, Y 25.6142, Z -110.0150, A 0, B 90, C 0, E1 0, E2 0, E3 0, E4 0 } C_DIS
LIN{ E6POS: X 709.1097, Y 26.1784, Z -110.0150, A 0, B 90, C 0, E1 0, E2 0, E3 0, E4 0 } C_DIS
LIN{ E6POS: X 709.1540, Y 27.1774, Z -110.0150, A 0, B 90, C 0, E1 0, E2 0, E3 0, E4 0 } C_DIS
LIN{ E6POS: X 709.1615, Y 27.3474, Z -110.0150, A 0, B 90, C 0, E1 0, E2 0, E3 0, E4 0 } C_DIS
LIN{ E6POS: X 709.2293, Y 28.3451, Z -110.0150, A 0, B 90, C 0, E1 0, E2 0, E3 0, E4 0 } C_DIS
LIN{ E6POS: X 709.2343, Y 28.4182, Z -110.0150, A 0, B 90, C 0, E1 0, E2 0, E3 0, E4 0 } C_DIS
LIN{ E6POS: X 709.2742, Y 29.4174, Z -110.0150, A 0, B 90, C 0, E1 0, E2 0, E3 0, E4 0 } C_DIS
LIN{ E6POS: X 709.2813, Y 29.5933, Z -110.0150, A 0, B 90, C 0, E1 0, E2 0, E3 0, E4 0 } C_DIS
LIN{ E6POS: X 709.3508, Y 30.5909, Z -110.0150, A 0, B 90, C 0, E1 0, E2 0, E3 0, E4 0 } C_DIS
LIN{ E6POS: X 709.3549, Y 30.6497, Z -110.0150, A 0, B 90, C 0, E1 0, E2 0, E3 0, E4 0 } C_DIS
LIN{ E6POS: X 709.3707, Y 31.5232, Z -110.0150, A 0, B 90, C 0, E1 0, E2 0, E3 0, E4 0 } C_DIS
LIN{ E6POS: X 709.3973, Y 32.1712, Z -110.0150, A 0, B 90, C 0, E1 0, E2 0, E3 0, E4 0 } C_DIS
LIN{ E6POS: X 709.4125, Y 33.1711, Z -110.0150, A 0, B 90, C 0, E1 0, E2 0, E3 0, E4 0 } C_DIS
LIN{ E6POS: X 709.4127, Y 33.1886, Z -110.0150, A 0, B 90, C 0, E1 0, E2 0, E3 0, E4 0 } C_DIS
LIN{ E6POS: X 709.4387, Y 33.9177, Z -110.0150, A 0, B 90, C 0, E1 0, E2 0, E3 0, E4 0 } C_DIS
LIN{ E6POS: X 709.4538, Y 34.9176, Z -110.0150, A 0, B 90, C 0, E1 0, E2 0, E3 0, E4 0 } C_DIS
LIN{ E6POS: X 709.4540, Y 34.9351, Z -110.0150, A 0, B 90, C 0, E1 0, E2 0, E3 0, E4 0 } C_DIS
LIN{ E6POS: X 709.4803, Y 35.6638, Z -110.0150, A 0, B 90, C 0, E1 0, E2 0, E3 0, E4 0 } C_DIS
LIN{ E6POS: X 709.4970, Y 36.5370, Z -110.0150, A 0, B 90, C 0, E1 0, E2 0, E3 0, E4 0 } C_DIS
LIN{ E6POS: X 709.5251, Y 37.1841, Z -110.0150, A 0, B 90, C 0, E1 0, E2 0, E3 0, E4 0 } C_DIS
LIN{ E6POS: X 709.5662, Y 38.1832, Z -110.0150, A 0, B 90, C 0, E1 0, E2 0, E3 0, E4 0 } C_DIS
LIN{ E6POS: X 709.5672, Y 38.2071, Z -110.0150, A 0, B 90, C 0, E1 0, E2 0, E3 0, E4 0 } C_DIS
LIN{ E6POS: X 709.6331, Y 39.0916, Z -110.0150, A 0, B 90, C 0, E1 0, E2 0, E3 0, E4 0 } C_DIS
LIN{ E6POS: X 709.6866, Y 40.0901, Z -110.0150, A 0, B 90, C 0, E1 0, E2 0, E3 0, E4 0 } C_DIS
LIN{ E6POS: X 709.6874, Y 40.1044, Z -110.0150, A 0, B 90, C 0, E1 0, E2 0, E3 0, E4 0 } C_DIS
LIN{ E6POS: X 709.7607, Y 40.9820, Z -110.0150, A 0, B 90, C 0, E1 0, E2 0, E3 0, E4 0 } C_DIS
LIN{ E6POS: X 709.7948, Y 41.8404, Z -110.0150, A 0, B 90, C 0, E1 0, E2 0, E3 0, E4 0 } C_DIS
LIN{ E6POS: X 709.8346, Y 42.4770, Z -110.0150, A 0, B 90, C 0, E1 0, E2 0, E3 0, E4 0 } C_DIS
LIN{ E6POS: X 709.8705, Y 43.4763, Z -110.0150, A 0, B 90, C 0, E1 0, E2 0, E3 0, E4 0 } C_DIS
LIN{ E6POS: X 709.8716, Y 43.5045, Z -110.0150, A 0, B 90, C 0, E1 0, E2 0, E3 0, E4 0 } C_DIS
LIN{ E6POS: X 709.9126, Y 44.2358, Z -110.0150, A 0, B 90, C 0, E1 0, E2 0, E3 0, E4 0 } C_DIS
LIN{ E6POS: X 709.9471, Y 45.2352, Z -110.0150, A 0, B 90, C 0, E1 0, E2 0, E3 0, E4 0 } C_DIS
LIN{ E6POS: X 709.9501, Y 45.3208, Z -110.0150, A 0, B 90, C 0, E1 0, E2 0, E3 0, E4 0 } C_DIS
LIN{ E6POS: X 709.9915, Y 46.0813, Z -110.0150, A 0, B 90, C 0, E1 0, E2 0, E3 0, E4 0 } C_DIS
LIN{ E6POS: X 710.0264, Y 47.0807, Z -110.0150, A 0, B 90, C 0, E1 0, E2 0, E3 0, E4 0 } C_DIS
LIN{ E6POS: X 710.0275, Y 47.1109, Z -110.0150, A 0, B 90, C 0, E1 0, E2 0, E3 0, E4 0 } C_DIS
LIN{ E6POS: X 710.0688, Y 47.8371, Z -110.0150, A 0, B 90, C 0, E1 0, E2 0, E3 0, E4 0 } C_DIS
LIN{ E6POS: X 710.1016, Y 48.6988, Z -110.0150, A 0, B 90, C 0, E1 0, E2 0, E3 0, E4 0 } C_DIS
LIN{ E6POS: X 710.1425, Y 49.3250, Z -110.0150, A 0, B 90, C 0, E1 0, E2 0, E3 0, E4 0 } C_DIS
LIN{ E6POS: X 710.1718, Y 50.0603, Z -110.0150, A 0, B 90, C 0, E1 0, E2 0, E3 0, E4 0 } C_DIS
LIN{ E6POS: X 710.2126, Y 50.6119, Z -110.0150, A 0, B 90, C 0, E1 0, E2 0, E3 0, E4 0 } C_DIS
LIN{ E6POS: X 710.2410, Y 51.2638, Z -110.0150, A 0, B 90, C 0, E1 0, E2 0, E3 0, E4 0 } C_DIS
LIN{ E6POS: X 710.2815, Y 51.7657, Z -110.0150, A 0, B 90, C 0, E1 0, E2 0, E3 0, E4 0 } C_DIS
LIN{ E6POS: X 710.3088, Y 52.3782, Z -110.0150, A 0, B 90, C 0, E1 0, E2 0, E3 0, E4 0 } C_DIS
LIN{ E6POS: X 710.3495, Y 52.8604, Z -110.0150, A 0, B 90, C 0, E1 0, E2 0, E3 0, E4 0 } C_DIS
LIN{ E6POS: X 710.9355, Y 52.7228, Z -110.0150, A 0, B 90, C 0, E1 0, E2 0, E3 0, E4 0 } C_DIS
LIN{ E6POS: X 711.3589, Y 52.6304, Z -110.0150, A 0, B 90, C 0, E1 0, E2 0, E3 0, E4 0 } C_DIS
LIN{ E6POS: X 712.3274, Y 52.3813, Z -110.0150, A 0, B 90, C 0, E1 0, E2 0, E3 0, E4 0 } C_DIS
LIN{ E6POS: X 713.1123, Y 52.1794, Z -110.0150, A 0, B 90, C 0, E1 0, E2 0, E3 0, E4 0 } C_DIS
LIN{ E6POS: X 714.0783, Y 51.9205, Z -110.0150, A 0, B 90, C 0, E1 0, E2 0, E3 0, E4 0 } C_DIS
LIN{ E6POS: X 714.3748, Y 51.8411, Z -110.0150, A 0, B 90, C 0, E1 0, E2 0, E3 0, E4 0 } C_DIS
LIN{ E6POS: X 715.3426, Y 51.5894, Z -110.0150, A 0, B 90, C 0, E1 0, E2 0, E3 0, E4 0 } C_DIS
LIN{ E6POS: X 716.3105, Y 51.3378, Z -110.0150, A 0, B 90, C 0, E1 0, E2 0, E3 0, E4 0 } C_DIS
LIN{ E6POS: X 717.2783, Y 51.0862, Z -110.0150, A 0, B 90, C 0, E1 0, E2 0, E3 0, E4 0 } C_DIS
LIN{ E6POS: X 717.8798, Y 50.9298, Z -110.0150, A 0, B 90, C 0, E1 0, E2 0, E3 0, E4 0 } C_DIS
LIN{ E6POS: X 718.8442, Y 50.6653, Z -110.0150, A 0, B 90, C 0, E1 0, E2 0, E3 0, E4 0 } C_DIS
LIN{ E6POS: X 719.8086, Y 50.4007, Z -110.0150, A 0, B 90, C 0, E1 0, E2 0, E3 0, E4 0 } C_DIS
LIN{ E6POS: X 720.4028, Y 50.2377, Z -110.0150, A 0, B 90, C 0, E1 0, E2 0, E3 0, E4 0 } C_DIS
LIN{ E6POS: X 721.3704, Y 49.9851, Z -110.0150, A 0, B 90, C 0, E1 0, E2 0, E3 0, E4 0 } C_DIS
LIN{ E6POS: X 722.3380, Y 49.7325, Z -110.0150, A 0, B 90, C 0, E1 0, E2 0, E3 0, E4 0 } C_DIS
LIN{ E6POS: X 723.3055, Y 49.4799, Z -110.0150, A 0, B 90, C 0, E1 0, E2 0, E3 0, E4 0 } C_DIS
LIN{ E6POS: X 724.2731, Y 49.2273, Z -110.0150, A 0, B 90, C 0, E1 0, E2 0, E3 0, E4 0 } C_DIS
LIN{ E6POS: X 725.2407, Y 48.9747, Z -110.0150, A 0, B 90, C 0, E1 0, E2 0, E3 0, E4 0 } C_DIS
LIN{ E6POS: X 726.2082, Y 48.7221, Z -110.0150, A 0, B 90, C 0, E1 0, E2 0, E3 0, E4 0 } C_DIS
LIN{ E6POS: X 726.2445, Y 48.7126, Z -110.0150, A 0, B 90, C 0, E1 0, E2 0, E3 0, E4 0 } C_DIS
LIN{ E6POS: X 727.2083, Y 48.4460, Z -110.0150, A 0, B 90, C 0, E1 0, E2 0, E3 0, E4 0 } C_DIS
LIN{ E6POS: X 728.1721, Y 48.1794, Z -110.0150, A 0, B 90, C 0, E1 0, E2 0, E3 0, E4 0 } C_DIS
LIN{ E6POS: X 729.1359, Y 47.9128, Z -110.0150, A 0, B 90, C 0, E1 0, E2 0, E3 0, E4 0 } C_DIS
LIN{ E6POS: X 730.0997, Y 47.6461, Z -110.0150, A 0, B 90, C 0, E1 0, E2 0, E3 0, E4 0 } C_DIS
LIN{ E6POS: X 730.4488, Y 47.5496, Z -110.0150, A 0, B 90, C 0, E1 0, E2 0, E3 0, E4 0 } C_DIS
LIN{ E6POS: X 731.4190, Y 47.3070, Z -110.0150, A 0, B 90, C 0, E1 0, E2 0, E3 0, E4 0 } C_DIS
LIN{ E6POS: X 732.3891, Y 47.0645, Z -110.0150, A 0, B 90, C 0, E1 0, E2 0, E3 0, E4 0 } C_DIS
LIN{ E6POS: X 733.3593, Y 46.8219, Z -110.0150, A 0, B 90, C 0, E1 0, E2 0, E3 0, E4 0 } C_DIS
LIN{ E6POS: X 734.3294, Y 46.5794, Z -110.0150, A 0, B 90, C 0, E1 0, E2 0, E3 0, E4 0 } C_DIS
LIN{ E6POS: X 735.2995, Y 46.3368, Z -110.0150, A 0, B 90, C 0, E1 0, E2 0, E3 0, E4 0 } C_DIS
LIN{ E6POS: X 736.2697, Y 46.0943, Z -110.0150, A 0, B 90, C 0, E1 0, E2 0, E3 0, E4 0 } C_DIS
LIN{ E6POS: X 737.2398, Y 45.8518, Z -110.0150, A 0, B 90, C 0, E1 0, E2 0, E3 0, E4 0 } C_DIS
LIN{ E6POS: X 737.6696, Y 45.7443, Z -110.0150, A 0, B 90, C 0, E1 0, E2 0, E3 0, E4 0 } C_DIS
LIN{ E6POS: X 738.6363, Y 45.4886, Z -110.0150, A 0, B 90, C 0, E1 0, E2 0, E3 0, E4 0 } C_DIS
LIN{ E6POS: X 739.6030, Y 45.2328, Z -110.0150, A 0, B 90, C 0, E1 0, E2 0, E3 0, E4 0 } C_DIS
LIN{ E6POS: X 740.5698, Y 44.9770, Z -110.0150, A 0, B 90, C 0, E1 0, E2 0, E3 0, E4 0 } C_DIS
LIN{ E6POS: X 741.5365, Y 44.7213, Z -110.0150, A 0, B 90, C 0, E1 0, E2 0, E3 0, E4 0 } C_DIS
LIN{ E6POS: X 742.5032, Y 44.4655, Z -110.0150, A 0, B 90, C 0, E1 0, E2 0, E3 0, E4 0 } C_DIS
LIN{ E6POS: X 742.8795, Y 44.3659, Z -110.0150, A 0, B 90, C 0, E1 0, E2 0, E3 0, E4 0 } C_DIS
LIN{ E6POS: X 743.8543, Y 44.1426, Z -110.0150, A 0, B 90, C 0, E1 0, E2 0, E3 0, E4 0 } C_DIS
LIN{ E6POS: X 744.8290, Y 43.9192, Z -110.0150, A 0, B 90, C 0, E1 0, E2 0, E3 0, E4 0 } C_DIS
LIN{ E6POS: X 745.8038, Y 43.6959, Z -110.0150, A 0, B 90, C 0, E1 0, E2 0, E3 0, E4 0 } C_DIS
LIN{ E6POS: X 746.7785, Y 43.4725, Z -110.0150, A 0, B 90, C 0, E1 0, E2 0, E3 0, E4 0 } C_DIS
LIN{ E6POS: X 747.7532, Y 43.2492, Z -110.0150, A 0, B 90, C 0, E1 0, E2 0, E3 0, E4 0 } C_DIS
LIN{ E6POS: X 748.7280, Y 43.0258, Z -110.0150, A 0, B 90, C 0, E1 0, E2 0, E3 0, E4 0 } C_DIS
LIN{ E6POS: X 749.7027, Y 42.8025, Z -110.0150, A 0, B 90, C 0, E1 0, E2 0, E3 0, E4 0 } C_DIS
LIN{ E6POS: X 750.5234, Y 42.6144, Z -110.0150, A 0, B 90, C 0, E1 0, E2 0, E3 0, E4 0 } C_DIS
LIN{ E6POS: X 751.4956, Y 42.3800, Z -110.0150, A 0, B 90, C 0, E1 0, E2 0, E3 0, E4 0 } C_DIS
LIN{ E6POS: X 752.4677, Y 42.1455, Z -110.0150, A 0, B 90, C 0, E1 0, E2 0, E3 0, E4 0 } C_DIS
LIN{ E6POS: X 753.4398, Y 41.9111, Z -110.0150, A 0, B 90, C 0, E1 0, E2 0, E3 0, E4 0 } C_DIS
LIN{ E6POS: X 754.4119, Y 41.6766, Z -110.0150, A 0, B 90, C 0, E1 0, E2 0, E3 0, E4 0 } C_DIS
LIN{ E6POS: X 755.3841, Y 41.4422, Z -110.0150, A 0, B 90, C 0, E1 0, E2 0, E3 0, E4 0 } C_DIS
LIN{ E6POS: X 756.0662, Y 41.2777, Z -110.0150, A 0, B 90, C 0, E1 0, E2 0, E3 0, E4 0 } C_DIS
LIN{ E6POS: X 757.0483, Y 41.0892, Z -110.0150, A 0, B 90, C 0, E1 0, E2 0, E3 0, E4 0 } C_DIS
LIN{ E6POS: X 758.0303, Y 40.9008, Z -110.0150, A 0, B 90, C 0, E1 0, E2 0, E3 0, E4 0 } C_DIS
LIN{ E6POS: X 759.0124, Y 40.7124, Z -110.0150, A 0, B 90, C 0, E1 0, E2 0, E3 0, E4 0 } C_DIS
LIN{ E6POS: X 759.9945, Y 40.5239, Z -110.0150, A 0, B 90, C 0, E1 0, E2 0, E3 0, E4 0 } C_DIS
LIN{ E6POS: X 760.9766, Y 40.3355, Z -110.0150, A 0, B 90, C 0, E1 0, E2 0, E3 0, E4 0 } C_DIS
LIN{ E6POS: X 761.9587, Y 40.1471, Z -110.0150, A 0, B 90, C 0, E1 0, E2 0, E3 0, E4 0 } C_DIS
LIN{ E6POS: X 762.9408, Y 39.9587, Z -110.0150, A 0, B 90, C 0, E1 0, E2 0, E3 0, E4 0 } C_DIS
LIN{ E6POS: X 763.1757, Y 39.9136, Z -110.0150, A 0, B 90, C 0, E1 0, E2 0, E3 0, E4 0 } C_DIS
LIN{ E6POS: X 764.1563, Y 39.7176, Z -110.0150, A 0, B 90, C 0, E1 0, E2 0, E3 0, E4 0 } C_DIS
LIN{ E6POS: X 765.1369, Y 39.5215, Z -110.0150, A 0, B 90, C 0, E1 0, E2 0, E3 0, E4 0 } C_DIS
LIN{ E6POS: X 766.1175, Y 39.3255, Z -110.0150, A 0, B 90, C 0, E1 0, E2 0, E3 0, E4 0 } C_DIS
LIN{ E6POS: X 767.0981, Y 39.1294, Z -110.0150, A 0, B 90, C 0, E1 0, E2 0, E3 0, E4 0 } C_DIS
LIN{ E6POS: X 768.0787, Y 38.9334, Z -110.0150, A 0, B 90, C 0, E1 0, E2 0, E3 0, E4 0 } C_DIS
LIN{ E6POS: X 768.3758, Y 38.8740, Z -110.0150, A 0, B 90, C 0, E1 0, E2 0, E3 0, E4 0 } C_DIS
LIN{ E6POS: X 769.3694, Y 38.7604, Z -110.0150, A 0, B 90, C 0, E1 0, E2 0, E3 0, E4 0 } C_DIS
LIN{ E6POS: X 770.3629, Y 38.6467, Z -110.0150, A 0, B 90, C 0, E1 0, E2 0, E3 0, E4 0 } C_DIS
LIN{ E6POS: X 771.3564, Y 38.5331, Z -110.0150, A 0, B 90, C 0, E1 0, E2 0, E3 0, E4 0 } C_DIS
LIN{ E6POS: X 772.3499, Y 38.4194, Z -110.0150, A 0, B 90, C 0, E1 0, E2 0, E3 0, E4 0 } C_DIS
LIN{ E6POS: X 773.3434, Y 38.3058, Z -110.0150, A 0, B 90, C 0, E1 0, E2 0, E3 0, E4 0 } C_DIS
LIN{ E6POS: X 773.9950, Y 38.2312, Z -110.0150, A 0, B 90, C 0, E1 0, E2 0, E3 0, E4 0 } C_DIS
LIN{ E6POS: X 774.9884, Y 38.1161, Z -110.0150, A 0, B 90, C 0, E1 0, E2 0, E3 0, E4 0 } C_DIS
LIN{ E6POS: X 775.9817, Y 38.0009, Z -110.0150, A 0, B 90, C 0, E1 0, E2 0, E3 0, E4 0 } C_DIS
LIN{ E6POS: X 776.9751, Y 37.8857, Z -110.0150, A 0, B 90, C 0, E1 0, E2 0, E3 0, E4 0 } C_DIS
LIN{ E6POS: X 777.9684, Y 37.7706, Z -110.0150, A 0, B 90, C 0, E1 0, E2 0, E3 0, E4 0 } C_DIS
LIN{ E6POS: X 778.1782, Y 37.7463, Z -110.0150, A 0, B 90, C 0, E1 0, E2 0, E3 0, E4 0 } C_DIS
LIN{ E6POS: X 779.1779, Y 37.7237, Z -110.0150, A 0, B 90, C 0, E1 0, E2 0, E3 0, E4 0 } C_DIS
LIN{ E6POS: X 780.1777, Y 37.7012, Z -110.0150, A 0, B 90, C 0, E1 0, E2 0, E3 0, E4 0 } C_DIS
LIN{ E6POS: X 781.1774, Y 37.6786, Z -110.0150, A 0, B 90, C 0, E1 0, E2 0, E3 0, E4 0 } C_DIS
LIN{ E6POS: X 782.1772, Y 37.6561, Z -110.0150, A 0, B 90, C 0, E1 0, E2 0, E3 0, E4 0 } C_DIS
LIN{ E6POS: X 782.6791, Y 37.6448, Z -110.0150, A 0, B 90, C 0, E1 0, E2 0, E3 0, E4 0 } C_DIS
LIN{ E6POS: X 783.6789, Y 37.6243, Z -110.0150, A 0, B 90, C 0, E1 0, E2 0, E3 0, E4 0 } C_DIS
LIN{ E6POS: X 784.6787, Y 37.6039, Z -110.0150, A 0, B 90, C 0, E1 0, E2 0, E3 0, E4 0 } C_DIS
LIN{ E6POS: X 785.6785, Y 37.5834, Z -110.0150, A 0, B 90, C 0, E1 0, E2 0, E3 0, E4 0 } C_DIS
LIN{ E6POS: X 786.0999, Y 37.5748, Z -110.0150, A 0, B 90, C 0, E1 0, E2 0, E3 0, E4 0 } C_DIS
LIN{ E6POS: X 787.0975, Y 37.6437, Z -110.0150, A 0, B 90, C 0, E1 0, E2 0, E3 0, E4 0 } C_DIS
LIN{ E6POS: X 788.0951, Y 37.7125, Z -110.0150, A 0, B 90, C 0, E1 0, E2 0, E3 0, E4 0 } C_DIS
LIN{ E6POS: X 789.0927, Y 37.7814, Z -110.0150, A 0, B 90, C 0, E1 0, E2 0, E3 0, E4 0 } C_DIS
LIN{ E6POS: X 789.8559, Y 37.8341, Z -110.0150, A 0, B 90, C 0, E1 0, E2 0, E3 0, E4 0 } C_DIS
LIN{ E6POS: X 790.8534, Y 37.9049, Z -110.0150, A 0, B 90, C 0, E1 0, E2 0, E3 0, E4 0 } C_DIS
LIN{ E6POS: X 791.8509, Y 37.9757, Z -110.0150, A 0, B 90, C 0, E1 0, E2 0, E3 0, E4 0 } C_DIS
LIN{ E6POS: X 792.7685, Y 38.0409, Z -110.0150, A 0, B 90, C 0, E1 0, E2 0, E3 0, E4 0 } C_DIS
LIN{ E6POS: X 793.7601, Y 38.1698, Z -110.0150, A 0, B 90, C 0, E1 0, E2 0, E3 0, E4 0 } C_DIS
LIN{ E6POS: X 794.7518, Y 38.2986, Z -110.0150, A 0, B 90, C 0, E1 0, E2 0, E3 0, E4 0 } C_DIS
LIN{ E6POS: X 795.7435, Y 38.4275, Z -110.0150, A 0, B 90, C 0, E1 0, E2 0, E3 0, E4 0 } C_DIS
LIN{ E6POS: X 796.1515, Y 38.4806, Z -110.0150, A 0, B 90, C 0, E1 0, E2 0, E3 0, E4 0 } C_DIS
LIN{ E6POS: X 797.1432, Y 38.6094, Z -110.0150, A 0, B 90, C 0, E1 0, E2 0, E3 0, E4 0 } C_DIS
LIN{ E6POS: X 798.1349, Y 38.7383, Z -110.0150, A 0, B 90, C 0, E1 0, E2 0, E3 0, E4 0 } C_DIS
LIN{ E6POS: X 798.8097, Y 38.8260, Z -110.0150, A 0, B 90, C 0, E1 0, E2 0, E3 0, E4 0 } C_DIS
LIN{ E6POS: X 798.7068, Y 37.8313, Z -110.0150, A 0, B 90, C 0, E1 0, E2 0, E3 0, E4 0 } C_DIS
LIN{ E6POS: X 798.6040, Y 36.8366, Z -110.0150, A 0, B 90, C 0, E1 0, E2 0, E3 0, E4 0 } C_DIS
LIN{ E6POS: X 798.5012, Y 35.8419, Z -110.0150, A 0, B 90, C 0, E1 0, E2 0, E3 0, E4 0 } C_DIS
LIN{ E6POS: X 798.3983, Y 34.8472, Z -110.0150, A 0, B 90, C 0, E1 0, E2 0, E3 0, E4 0 } C_DIS
LIN{ E6POS: X 798.2955, Y 33.8525, Z -110.0150, A 0, B 90, C 0, E1 0, E2 0, E3 0, E4 0 } C_DIS
LIN{ E6POS: X 798.1927, Y 32.8578, Z -110.0150, A 0, B 90, C 0, E1 0, E2 0, E3 0, E4 0 } C_DIS
LIN{ E6POS: X 798.0898, Y 31.8631, Z -110.0150, A 0, B 90, C 0, E1 0, E2 0, E3 0, E4 0 } C_DIS
LIN{ E6POS: X 797.9870, Y 30.8684, Z -110.0150, A 0, B 90, C 0, E1 0, E2 0, E3 0, E4 0 } C_DIS
LIN{ E6POS: X 797.8842, Y 29.8737, Z -110.0150, A 0, B 90, C 0, E1 0, E2 0, E3 0, E4 0 } C_DIS
LIN{ E6POS: X 797.8648, Y 29.6863, Z -110.0150, A 0, B 90, C 0, E1 0, E2 0, E3 0, E4 0 } C_DIS
LIN{ E6POS: X 797.7620, Y 28.6916, Z -110.0150, A 0, B 90, C 0, E1 0, E2 0, E3 0, E4 0 } C_DIS
LIN{ E6POS: X 797.6591, Y 27.6969, Z -110.0150, A 0, B 90, C 0, E1 0, E2 0, E3 0, E4 0 } C_DIS
LIN{ E6POS: X 797.5563, Y 26.7022, Z -110.0150, A 0, B 90, C 0, E1 0, E2 0, E3 0, E4 0 } C_DIS
LIN{ E6POS: X 797.4535, Y 25.7075, Z -110.0150, A 0, B 90, C 0, E1 0, E2 0, E3 0, E4 0 } C_DIS
LIN{ E6POS: X 797.3506, Y 24.7128, Z -110.0150, A 0, B 90, C 0, E1 0, E2 0, E3 0, E4 0 } C_DIS
LIN{ E6POS: X 797.2478, Y 23.7181, Z -110.0150, A 0, B 90, C 0, E1 0, E2 0, E3 0, E4 0 } C_DIS
LIN{ E6POS: X 797.1450, Y 22.7234, Z -110.0150, A 0, B 90, C 0, E1 0, E2 0, E3 0, E4 0 } C_DIS
LIN{ E6POS: X 797.1224, Y 22.5051, Z -108.0150, A 0, B 90, C 0, E1 0, E2 0, E3 0, E4 0 } C_DIS
LIN{ E6POS: X 797.0002, Y 21.5126, Z -108.0150, A 0, B 90, C 0, E1 0, E2 0, E3 0, E4 0 } C_DIS
LIN{ E6POS: X 796.8780, Y 20.5201, Z -108.0150, A 0, B 90, C 0, E1 0, E2 0, E3 0, E4 0 } C_DIS
LIN{ E6POS: X 796.7559, Y 19.5276, Z -108.0150, A 0, B 90, C 0, E1 0, E2 0, E3 0, E4 0 } C_DIS
LIN{ E6POS: X 796.6337, Y 18.5351, Z -108.0150, A 0, B 90, C 0, E1 0, E2 0, E3 0, E4 0 } C_DIS
LIN{ E6POS: X 796.5115, Y 17.5426, Z -108.0150, A 0, B 90, C 0, E1 0, E2 0, E3 0, E4 0 } C_DIS
LIN{ E6POS: X 796.3893, Y 16.5500, Z -108.0150, A 0, B 90, C 0, E1 0, E2 0, E3 0, E4 0 } C_DIS
LIN{ E6POS: X 796.2672, Y 15.5575, Z -108.0150, A 0, B 90, C 0, E1 0, E2 0, E3 0, E4 0 } C_DIS
LIN{ E6POS: X 796.1450, Y 14.5650, Z -108.0150, A 0, B 90, C 0, E1 0, E2 0, E3 0, E4 0 } C_DIS
LIN{ E6POS: X 796.0228, Y 13.5725, Z -108.0150, A 0, B 90, C 0, E1 0, E2 0, E3 0, E4 0 } C_DIS
LIN{ E6POS: X 795.9281, Y 12.8028, Z -108.0150, A 0, B 90, C 0, E1 0, E2 0, E3 0, E4 0 } C_DIS
LIN{ E6POS: X 795.8059, Y 11.8103, Z -108.0150, A 0, B 90, C 0, E1 0, E2 0, E3 0, E4 0 } C_DIS
LIN{ E6POS: X 795.6837, Y 10.8178, Z -108.0150, A 0, B 90, C 0, E1 0, E2 0, E3 0, E4 0 } C_DIS
LIN{ E6POS: X 795.5615, Y 9.8253, Z -108.0150, A 0, B 90, C 0, E1 0, E2 0, E3 0, E4 0 } C_DIS
LIN{ E6POS: X 795.4393, Y 8.8328, Z -108.0150, A 0, B 90, C 0, E1 0, E2 0, E3 0, E4 0 } C_DIS
LIN{ E6POS: X 795.3172, Y 7.8402, Z -108.0150, A 0, B 90, C 0, E1 0, E2 0, E3 0, E4 0 } C_DIS
LIN{ E6POS: X 795.2562, Y 7.3452, Z -108.0150, A 0, B 90, C 0, E1 0, E2 0, E3 0, E4 0 } C_DIS
LIN{ E6POS: X 795.0854, Y 6.3599, Z -108.0150, A 0, B 90, C 0, E1 0, E2 0, E3 0, E4 0 } C_DIS
LIN{ E6POS: X 794.9146, Y 5.3746, Z -108.0150, A 0, B 90, C 0, E1 0, E2 0, E3 0, E4 0 } C_DIS
LIN{ E6POS: X 794.7438, Y 4.3893, Z -108.0150, A 0, B 90, C 0, E1 0, E2 0, E3 0, E4 0 } C_DIS
LIN{ E6POS: X 794.5730, Y 3.4040, Z -108.0150, A 0, B 90, C 0, E1 0, E2 0, E3 0, E4 0 } C_DIS
LIN{ E6POS: X 794.4021, Y 2.4187, Z -108.0150, A 0, B 90, C 0, E1 0, E2 0, E3 0, E4 0 } C_DIS
LIN{ E6POS: X 794.2313, Y 1.4334, Z -108.0150, A 0, B 90, C 0, E1 0, E2 0, E3 0, E4 0 } C_DIS
LIN{ E6POS: X 794.0605, Y 0.4481, Z -108.0150, A 0, B 90, C 0, E1 0, E2 0, E3 0, E4 0 } C_DIS
LIN{ E6POS: X 793.8897, Y -0.5372, Z -108.0150, A 0, B 90, C 0, E1 0, E2 0, E3 0, E4 0 } C_DIS
LIN{ E6POS: X 793.8321, Y -0.8693, Z -108.0150, A 0, B 90, C 0, E1 0, E2 0, E3 0, E4 0 } C_DIS
LIN{ E6POS: X 793.6613, Y -1.8546, Z -108.0150, A 0, B 90, C 0, E1 0, E2 0, E3 0, E4 0 } C_DIS
LIN{ E6POS: X 793.4905, Y -2.8399, Z -108.0150, A 0, B 90, C 0, E1 0, E2 0, E3 0, E4 0 } C_DIS
LIN{ E6POS: X 793.3196, Y -3.8252, Z -108.0150, A 0, B 90, C 0, E1 0, E2 0, E3 0, E4 0 } C_DIS
LIN{ E6POS: X 793.1488, Y -4.8106, Z -108.0150, A 0, B 90, C 0, E1 0, E2 0, E3 0, E4 0 } C_DIS
LIN{ E6POS: X 793.0310, Y -5.4900, Z -108.0150, A 0, B 90, C 0, E1 0, E2 0, E3 0, E4 0 } C_DIS
LIN{ E6POS: X 792.7476, Y -6.4490, Z -108.0150, A 0, B 90, C 0, E1 0, E2 0, E3 0, E4 0 } C_DIS
LIN{ E6POS: X 792.4642, Y -7.4080, Z -108.0150, A 0, B 90, C 0, E1 0, E2 0, E3 0, E4 0 } C_DIS
LIN{ E6POS: X 792.1808, Y -8.3670, Z -108.0150, A 0, B 90, C 0, E1 0, E2 0, E3 0, E4 0 } C_DIS
LIN{ E6POS: X 791.8974, Y -9.3260, Z -108.0150, A 0, B 90, C 0, E1 0, E2 0, E3 0, E4 0 } C_DIS
LIN{ E6POS: X 791.6139, Y -10.2850, Z -108.0150, A 0, B 90, C 0, E1 0, E2 0, E3 0, E4 0 } C_DIS
LIN{ E6POS: X 791.3305, Y -11.2440, Z -108.0150, A 0, B 90, C 0, E1 0, E2 0, E3 0, E4 0 } C_DIS
LIN{ E6POS: X 791.2628, Y -11.4732, Z -108.0150, A 0, B 90, C 0, E1 0, E2 0, E3 0, E4 0 } C_DIS
LIN{ E6POS: X 790.9794, Y -12.4322, Z -108.0150, A 0, B 90, C 0, E1 0, E2 0, E3 0, E4 0 } C_DIS
LIN{ E6POS: X 790.6959, Y -13.3912, Z -108.0150, A 0, B 90, C 0, E1 0, E2 0, E3 0, E4 0 } C_DIS
LIN{ E6POS: X 790.4125, Y -14.3502, Z -108.0150, A 0, B 90, C 0, E1 0, E2 0, E3 0, E4 0 } C_DIS
LIN{ E6POS: X 790.2681, Y -14.8387, Z -108.0150, A 0, B 90, C 0, E1 0, E2 0, E3 0, E4 0 } C_DIS
LIN{ E6POS: X 789.6733, Y -15.6426, Z -108.0150, A 0, B 90, C 0, E1 0, E2 0, E3 0, E4 0 } C_DIS
LIN{ E6POS: X 789.0784, Y -16.4464, Z -108.0150, A 0, B 90, C 0, E1 0, E2 0, E3 0, E4 0 } C_DIS
LIN{ E6POS: X 788.4835, Y -17.2502, Z -108.0150, A 0, B 90, C 0, E1 0, E2 0, E3 0, E4 0 } C_DIS
LIN{ E6POS: X 788.0411, Y -17.8480, Z -108.0150, A 0, B 90, C 0, E1 0, E2 0, E3 0, E4 0 } C_DIS
LIN{ E6POS: X 787.4463, Y -18.6519, Z -108.0150, A 0, B 90, C 0, E1 0, E2 0, E3 0, E4 0 } C_DIS
LIN{ E6POS: X 786.8514, Y -19.4557, Z -108.0150, A 0, B 90, C 0, E1 0, E2 0, E3 0, E4 0 } C_DIS
LIN{ E6POS: X 786.7884, Y -19.5408, Z -108.0150, A 0, B 90, C 0, E1 0, E2 0, E3 0, E4 0 } C_DIS
LIN{ E6POS: X 785.8312, Y -19.8300, Z -108.0150, A 0, B 90, C 0, E1 0, E2 0, E3 0, E4 0 } C_DIS
LIN{ E6POS: X 784.8739, Y -20.1192, Z -108.0150, A 0, B 90, C 0, E1 0, E2 0, E3 0, E4 0 } C_DIS
LIN{ E6POS: X 783.9561, Y -20.3965, Z -108.0150, A 0, B 90, C 0, E1 0, E2 0, E3 0, E4 0 } C_DIS
LIN{ E6POS: X 783.0001, Y -20.6896, Z -108.0150, A 0, B 90, C 0, E1 0, E2 0, E3 0, E4 0 } C_DIS
LIN{ E6POS: X 782.3841, Y -20.8785, Z -108.0150, A 0, B 90, C 0, E1 0, E2 0, E3 0, E4 0 } C_DIS
LIN{ E6POS: X 781.3933, Y -20.7436, Z -108.0150, A 0, B 90, C 0, E1 0, E2 0, E3 0, E4 0 } C_DIS
LIN{ E6POS: X 780.4321, Y -20.6127, Z -108.0150, A 0, B 90, C 0, E1 0, E2 0, E3 0, E4 0 } C_DIS
LIN{ E6POS: X 779.4408, Y -20.4811, Z -108.0150, A 0, B 90, C 0, E1 0, E2 0, E3 0, E4 0 } C_DIS
LIN{ E6POS: X 778.4495, Y -20.3495, Z -108.0150, A 0, B 90, C 0, E1 0, E2 0, E3 0, E4 0 } C_DIS
LIN{ E6POS: X 777.4582, Y -20.2179, Z -108.0150, A 0, B 90, C 0, E1 0, E2 0, E3 0, E4 0 } C_DIS
LIN{ E6POS: X 776.8499, Y -20.1371, Z -108.0150, A 0, B 90, C 0, E1 0, E2 0, E3 0, E4 0 } C_DIS
LIN{ E6POS: X 775.8754, Y -19.9130, Z -108.0150, A 0, B 90, C 0, E1 0, E2 0, E3 0, E4 0 } C_DIS
LIN{ E6POS: X 774.9008, Y -19.6889, Z -108.0150, A 0, B 90, C 0, E1 0, E2 0, E3 0, E4 0 } C_DIS
LIN{ E6POS: X 774.4570, Y -19.5869, Z -108.0150, A 0, B 90, C 0, E1 0, E2 0, E3 0, E4 0 } C_DIS
LIN{ E6POS: X 773.4804, Y -19.3720, Z -108.0150, A 0, B 90, C 0, E1 0, E2 0, E3 0, E4 0 } C_DIS
LIN{ E6POS: X 772.5037, Y -19.1571, Z -108.0150, A 0, B 90, C 0, E1 0, E2 0, E3 0, E4 0 } C_DIS
LIN{ E6POS: X 771.5271, Y -18.9422, Z -108.0150, A 0, B 90, C 0, E1 0, E2 0, E3 0, E4 0 } C_DIS
LIN{ E6POS: X 770.5504, Y -18.7274, Z -108.0150, A 0, B 90, C 0, E1 0, E2 0, E3 0, E4 0 } C_DIS
LIN{ E6POS: X 769.9781, Y -18.6015, Z -108.0150, A 0, B 90, C 0, E1 0, E2 0, E3 0, E4 0 } C_DIS
LIN{ E6POS: X 768.9863, Y -18.4738, Z -108.0150, A 0, B 90, C 0, E1 0, E2 0, E3 0, E4 0 } C_DIS
LIN{ E6POS: X 767.9944, Y -18.3461, Z -108.0150, A 0, B 90, C 0, E1 0, E2 0, E3 0, E4 0 } C_DIS
LIN{ E6POS: X 767.0830, Y -18.2288, Z -108.0150, A 0, B 90, C 0, E1 0, E2 0, E3 0, E4 0 } C_DIS
LIN{ E6POS: X 766.0904, Y -18.1077, Z -108.0150, A 0, B 90, C 0, E1 0, E2 0, E3 0, E4 0 } C_DIS
LIN{ E6POS: X 765.0977, Y -17.9866, Z -108.0150, A 0, B 90, C 0, E1 0, E2 0, E3 0, E4 0 } C_DIS
LIN{ E6POS: X 764.1051, Y -17.8654, Z -108.0150, A 0, B 90, C 0, E1 0, E2 0, E3 0, E4 0 } C_DIS
LIN{ E6POS: X 763.1125, Y -17.7443, Z -108.0150, A 0, B 90, C 0, E1 0, E2 0, E3 0, E4 0 } C_DIS
LIN{ E6POS: X 762.1198, Y -17.6231, Z -108.0150, A 0, B 90, C 0, E1 0, E2 0, E3 0, E4 0 } C_DIS
LIN{ E6POS: X 761.5624, Y -17.5551, Z -108.0150, A 0, B 90, C 0, E1 0, E2 0, E3 0, E4 0 } C_DIS
LIN{ E6POS: X 760.5646, Y -17.4880, Z -108.0150, A 0, B 90, C 0, E1 0, E2 0, E3 0, E4 0 } C_DIS
LIN{ E6POS: X 759.5669, Y -17.4208, Z -108.0150, A 0, B 90, C 0, E1 0, E2 0, E3 0, E4 0 } C_DIS
LIN{ E6POS: X 758.5691, Y -17.3537, Z -108.0150, A 0, B 90, C 0, E1 0, E2 0, E3 0, E4 0 } C_DIS
LIN{ E6POS: X 758.5187, Y -17.3503, Z -108.0150, A 0, B 90, C 0, E1 0, E2 0, E3 0, E4 0 } C_DIS
LIN{ E6POS: X 757.5208, Y -17.2856, Z -108.0150, A 0, B 90, C 0, E1 0, E2 0, E3 0, E4 0 } C_DIS
LIN{ E6POS: X 756.5229, Y -17.2209, Z -108.0150, A 0, B 90, C 0, E1 0, E2 0, E3 0, E4 0 } C_DIS
LIN{ E6POS: X 755.5250, Y -17.1561, Z -108.0150, A 0, B 90, C 0, E1 0, E2 0, E3 0, E4 0 } C_DIS
LIN{ E6POS: X 754.5271, Y -17.0914, Z -108.0150, A 0, B 90, C 0, E1 0, E2 0, E3 0, E4 0 } C_DIS
LIN{ E6POS: X 753.5292, Y -17.0267, Z -108.0150, A 0, B 90, C 0, E1 0, E2 0, E3 0, E4 0 } C_DIS
LIN{ E6POS: X 752.6590, Y -16.9702, Z -108.0150, A 0, B 90, C 0, E1 0, E2 0, E3 0, E4 0 } C_DIS
LIN{ E6POS: X 751.6592, Y -16.9540, Z -108.0150, A 0, B 90, C 0, E1 0, E2 0, E3 0, E4 0 } C_DIS
LIN{ E6POS: X 750.6593, Y -16.9377, Z -108.0150, A 0, B 90, C 0, E1 0, E2 0, E3 0, E4 0 } C_DIS
LIN{ E6POS: X 749.8194, Y -16.9241, Z -108.0150, A 0, B 90, C 0, E1 0, E2 0, E3 0, E4 0 } C_DIS
LIN{ E6POS: X 748.8195, Y -16.9052, Z -108.0150, A 0, B 90, C 0, E1 0, E2 0, E3 0, E4 0 } C_DIS
LIN{ E6POS: X 747.8197, Y -16.8863, Z -108.0150, A 0, B 90, C 0, E1 0, E2 0, E3 0, E4 0 } C_DIS
LIN{ E6POS: X 746.8199, Y -16.8674, Z -108.0150, A 0, B 90, C 0, E1 0, E2 0, E3 0, E4 0 } C_DIS
LIN{ E6POS: X 745.8201, Y -16.8485, Z -108.0150, A 0, B 90, C 0, E1 0, E2 0, E3 0, E4 0 } C_DIS
LIN{ E6POS: X 744.8203, Y -16.8296, Z -108.0150, A 0, B 90, C 0, E1 0, E2 0, E3 0, E4 0 } C_DIS
LIN{ E6POS: X 744.3233, Y -16.8202, Z -108.0150, A 0, B 90, C 0, E1 0, E2 0, E3 0, E4 0 } C_DIS
LIN{ E6POS: X 743.3243, Y -16.8649, Z -108.0150, A 0, B 90, C 0, E1 0, E2 0, E3 0, E4 0 } C_DIS
LIN{ E6POS: X 742.3253, Y -16.9097, Z -108.0150, A 0, B 90, C 0, E1 0, E2 0, E3 0, E4 0 } C_DIS
LIN{ E6POS: X 742.0410, Y -16.9224, Z -108.0150, A 0, B 90, C 0, E1 0, E2 0, E3 0, E4 0 } C_DIS
LIN{ E6POS: X 741.0416, Y -16.9570, Z -108.0150, A 0, B 90, C 0, E1 0, E2 0, E3 0, E4 0 } C_DIS
LIN{ E6POS: X 740.0422, Y -16.9916, Z -108.0150, A 0, B 90, C 0, E1 0, E2 0, E3 0, E4 0 } C_DIS
LIN{ E6POS: X 739.0428, Y -17.0262, Z -108.0150, A 0, B 90, C 0, E1 0, E2 0, E3 0, E4 0 } C_DIS
LIN{ E6POS: X 738.0434, Y -17.0608, Z -108.0150, A 0, B 90, C 0, E1 0, E2 0, E3 0, E4 0 } C_DIS
LIN{ E6POS: X 737.6121, Y -17.0757, Z -108.0150, A 0, B 90, C 0, E1 0, E2 0, E3 0, E4 0 } C_DIS
LIN{ E6POS: X 736.6273, Y -17.2490, Z -108.0150, A 0, B 90, C 0, E1 0, E2 0, E3 0, E4 0 } C_DIS
LIN{ E6POS: X 736.2397, Y -17.3171, Z -108.0150, A 0, B 90, C 0, E1 0, E2 0, E3 0, E4 0 } C_DIS
LIN{ E6POS: X 735.2505, Y -17.4637, Z -108.0150, A 0, B 90, C 0, E1 0, E2 0, E3 0, E4 0 } C_DIS
LIN{ E6POS: X 734.2613, Y -17.6102, Z -108.0150, A 0, B 90, C 0, E1 0, E2 0, E3 0, E4 0 } C_DIS
LIN{ E6POS: X 733.5811, Y -17.7110, Z -108.0150, A 0, B 90, C 0, E1 0, E2 0, E3 0, E4 0 } C_DIS
LIN{ E6POS: X 733.1199, Y -18.0829, Z -108.0150, A 0, B 90, C 0, E1 0, E2 0, E3 0, E4 0 } C_DIS
LIN{ E6POS: X 732.3036, Y -18.6606, Z -108.0150, A 0, B 90, C 0, E1 0, E2 0, E3 0, E4 0 } C_DIS
LIN{ E6POS: X 732.2310, Y -18.7119, Z -108.0150, A 0, B 90, C 0, E1 0, E2 0, E3 0, E4 0 } C_DIS
LIN{ E6POS: X 732.9476, Y -19.4094, Z -108.0150, A 0, B 90, C 0, E1 0, E2 0, E3 0, E4 0 } C_DIS
LIN{ E6POS: X 733.1119, Y -19.5693, Z -108.0150, A 0, B 90, C 0, E1 0, E2 0, E3 0, E4 0 } C_DIS
LIN{ E6POS: X 733.5625, Y -20.0649, Z -108.0150, A 0, B 90, C 0, E1 0, E2 0, E3 0, E4 0 } C_DIS
LIN{ E6POS: X 734.4884, Y -20.4428, Z -108.0150, A 0, B 90, C 0, E1 0, E2 0, E3 0, E4 0 } C_DIS
LIN{ E6POS: X 735.4142, Y -20.8208, Z -108.0150, A 0, B 90, C 0, E1 0, E2 0, E3 0, E4 0 } C_DIS
LIN{ E6POS: X 736.2129, Y -21.1468, Z -108.0150, A 0, B 90, C 0, E1 0, E2 0, E3 0, E4 0 } C_DIS
LIN{ E6POS: X 737.1254, Y -21.5559, Z -108.0150, A 0, B 90, C 0, E1 0, E2 0, E3 0, E4 0 } C_DIS
LIN{ E6POS: X 737.5759, Y -21.7579, Z -108.0150, A 0, B 90, C 0, E1 0, E2 0, E3 0, E4 0 } C_DIS
LIN{ E6POS: X 738.5352, Y -22.0402, Z -108.0150, A 0, B 90, C 0, E1 0, E2 0, E3 0, E4 0 } C_DIS
LIN{ E6POS: X 739.4945, Y -22.3226, Z -108.0150, A 0, B 90, C 0, E1 0, E2 0, E3 0, E4 0 } C_DIS
LIN{ E6POS: X 740.4539, Y -22.6049, Z -108.0150, A 0, B 90, C 0, E1 0, E2 0, E3 0, E4 0 } C_DIS
LIN{ E6POS: X 741.4132, Y -22.8873, Z -108.0150, A 0, B 90, C 0, E1 0, E2 0, E3 0, E4 0 } C_DIS
LIN{ E6POS: X 741.9949, Y -23.0585, Z -108.0150, A 0, B 90, C 0, E1 0, E2 0, E3 0, E4 0 } C_DIS
LIN{ E6POS: X 742.9484, Y -23.3596, Z -108.0150, A 0, B 90, C 0, E1 0, E2 0, E3 0, E4 0 } C_DIS
LIN{ E6POS: X 743.9020, Y -23.6607, Z -108.0150, A 0, B 90, C 0, E1 0, E2 0, E3 0, E4 0 } C_DIS
LIN{ E6POS: X 744.2712, Y -23.7773, Z -108.0150, A 0, B 90, C 0, E1 0, E2 0, E3 0, E4 0 } C_DIS
LIN{ E6POS: X 745.2436, Y -24.0107, Z -108.0150, A 0, B 90, C 0, E1 0, E2 0, E3 0, E4 0 } C_DIS
LIN{ E6POS: X 746.2159, Y -24.2441, Z -108.0150, A 0, B 90, C 0, E1 0, E2 0, E3 0, E4 0 } C_DIS
LIN{ E6POS: X 747.1883, Y -24.4775, Z -108.0150, A 0, B 90, C 0, E1 0, E2 0, E3 0, E4 0 } C_DIS
LIN{ E6POS: X 748.1607, Y -24.7110, Z -108.0150, A 0, B 90, C 0, E1 0, E2 0, E3 0, E4 0 } C_DIS
LIN{ E6POS: X 749.1331, Y -24.9444, Z -108.0150, A 0, B 90, C 0, E1 0, E2 0, E3 0, E4 0 } C_DIS
LIN{ E6POS: X 749.7583, Y -25.0945, Z -108.0150, A 0, B 90, C 0, E1 0, E2 0, E3 0, E4 0 } C_DIS
LIN{ E6POS: X 750.7276, Y -25.3403, Z -108.0150, A 0, B 90, C 0, E1 0, E2 0, E3 0, E4 0 } C_DIS
LIN{ E6POS: X 751.6970, Y -25.5860, Z -108.0150, A 0, B 90, C 0, E1 0, E2 0, E3 0, E4 0 } C_DIS
LIN{ E6POS: X 752.5951, Y -25.8137, Z -108.0150, A 0, B 90, C 0, E1 0, E2 0, E3 0, E4 0 } C_DIS
LIN{ E6POS: X 753.5769, Y -26.0037, Z -108.0150, A 0, B 90, C 0, E1 0, E2 0, E3 0, E4 0 } C_DIS
LIN{ E6POS: X 754.5586, Y -26.1937, Z -108.0150, A 0, B 90, C 0, E1 0, E2 0, E3 0, E4 0 } C_DIS
LIN{ E6POS: X 755.5404, Y -26.3837, Z -108.0150, A 0, B 90, C 0, E1 0, E2 0, E3 0, E4 0 } C_DIS
LIN{ E6POS: X 756.5222, Y -26.5737, Z -108.0150, A 0, B 90, C 0, E1 0, E2 0, E3 0, E4 0 } C_DIS
LIN{ E6POS: X 757.5040, Y -26.7636, Z -108.0150, A 0, B 90, C 0, E1 0, E2 0, E3 0, E4 0 } C_DIS
LIN{ E6POS: X 758.4492, Y -26.9465, Z -108.0150, A 0, B 90, C 0, E1 0, E2 0, E3 0, E4 0 } C_DIS
LIN{ E6POS: X 759.4295, Y -27.1437, Z -108.0150, A 0, B 90, C 0, E1 0, E2 0, E3 0, E4 0 } C_DIS
LIN{ E6POS: X 760.4099, Y -27.3409, Z -108.0150, A 0, B 90, C 0, E1 0, E2 0, E3 0, E4 0 } C_DIS
LIN{ E6POS: X 761.3902, Y -27.5381, Z -108.0150, A 0, B 90, C 0, E1 0, E2 0, E3 0, E4 0 } C_DIS
LIN{ E6POS: X 761.4925, Y -27.5587, Z -108.0150, A 0, B 90, C 0, E1 0, E2 0, E3 0, E4 0 } C_DIS
LIN{ E6POS: X 762.4835, Y -27.6927, Z -108.0150, A 0, B 90, C 0, E1 0, E2 0, E3 0, E4 0 } C_DIS
LIN{ E6POS: X 763.4745, Y -27.8267, Z -108.0150, A 0, B 90, C 0, E1 0, E2 0, E3 0, E4 0 } C_DIS
LIN{ E6POS: X 764.4654, Y -27.9608, Z -108.0150, A 0, B 90, C 0, E1 0, E2 0, E3 0, E4 0 } C_DIS
LIN{ E6POS: X 765.4564, Y -28.0948, Z -108.0150, A 0, B 90, C 0, E1 0, E2 0, E3 0, E4 0 } C_DIS
LIN{ E6POS: X 766.4474, Y -28.2288, Z -108.0150, A 0, B 90, C 0, E1 0, E2 0, E3 0, E4 0 } C_DIS
LIN{ E6POS: X 767.0113, Y -28.3051, Z -108.0150, A 0, B 90, C 0, E1 0, E2 0, E3 0, E4 0 } C_DIS
LIN{ E6POS: X 768.0021, Y -28.4411, Z -108.0150, A 0, B 90, C 0, E1 0, E2 0, E3 0, E4 0 } C_DIS
LIN{ E6POS: X 768.9928, Y -28.5770, Z -108.0150, A 0, B 90, C 0, E1 0, E2 0, E3 0, E4 0 } C_DIS
LIN{ E6POS: X 769.9088, Y -28.7028, Z -108.0150, A 0, B 90, C 0, E1 0, E2 0, E3 0, E4 0 } C_DIS
LIN{ E6POS: X 770.9081, Y -28.7383, Z -108.0150, A 0, B 90, C 0, E1 0, E2 0, E3 0, E4 0 } C_DIS
LIN{ E6POS: X 771.9075, Y -28.7738, Z -108.0150, A 0, B 90, C 0, E1 0, E2 0, E3 0, E4 0 } C_DIS
LIN{ E6POS: X 772.9069, Y -28.8093, Z -108.0150, A 0, B 90, C 0, E1 0, E2 0, E3 0, E4 0 } C_DIS
LIN{ E6POS: X 773.9062, Y -28.8449, Z -108.0150, A 0, B 90, C 0, E1 0, E2 0, E3 0, E4 0 } C_DIS
LIN{ E6POS: X 774.3928, Y -28.8621, Z -108.0150, A 0, B 90, C 0, E1 0, E2 0, E3 0, E4 0 } C_DIS
LIN{ E6POS: X 775.3923, Y -28.8938, Z -108.0150, A 0, B 90, C 0, E1 0, E2 0, E3 0, E4 0 } C_DIS
LIN{ E6POS: X 776.3918, Y -28.9255, Z -108.0150, A 0, B 90, C 0, E1 0, E2 0, E3 0, E4 0 } C_DIS
LIN{ E6POS: X 776.7904, Y -28.9382, Z -108.0150, A 0, B 90, C 0, E1 0, E2 0, E3 0, E4 0 } C_DIS
LIN{ E6POS: X 777.7735, Y -29.1211, Z -108.0150, A 0, B 90, C 0, E1 0, E2 0, E3 0, E4 0 } C_DIS
LIN{ E6POS: X 778.7567, Y -29.3040, Z -108.0150, A 0, B 90, C 0, E1 0, E2 0, E3 0, E4 0 } C_DIS
LIN{ E6POS: X 779.7398, Y -29.4869, Z -108.0150, A 0, B 90, C 0, E1 0, E2 0, E3 0, E4 0 } C_DIS
LIN{ E6POS: X 780.1204, Y -29.5577, Z -108.0150, A 0, B 90, C 0, E1 0, E2 0, E3 0, E4 0 } C_DIS
LIN{ E6POS: X 781.1030, Y -29.7433, Z -108.0150, A 0, B 90, C 0, E1 0, E2 0, E3 0, E4 0 } C_DIS
LIN{ E6POS: X 781.9313, Y -29.8997, Z -108.0150, A 0, B 90, C 0, E1 0, E2 0, E3 0, E4 0 } C_DIS
LIN{ E6POS: X 782.6263, Y -30.6188, Z -108.0150, A 0, B 90, C 0, E1 0, E2 0, E3 0, E4 0 } C_DIS
LIN{ E6POS: X 783.3212, Y -31.3379, Z -108.0150, A 0, B 90, C 0, E1 0, E2 0, E3 0, E4 0 } C_DIS
LIN{ E6POS: X 783.9906, Y -32.0305, Z -108.0150, A 0, B 90, C 0, E1 0, E2 0, E3 0, E4 0 } C_DIS
LIN{ E6POS: X 784.6797, Y -32.7551, Z -108.0150, A 0, B 90, C 0, E1 0, E2 0, E3 0, E4 0 } C_DIS
LIN{ E6POS: X 785.1281, Y -33.2266, Z -108.0150, A 0, B 90, C 0, E1 0, E2 0, E3 0, E4 0 } C_DIS
LIN{ E6POS: X 785.2695, Y -34.2166, Z -108.0150, A 0, B 90, C 0, E1 0, E2 0, E3 0, E4 0 } C_DIS
LIN{ E6POS: X 785.4109, Y -35.2065, Z -108.0150, A 0, B 90, C 0, E1 0, E2 0, E3 0, E4 0 } C_DIS
LIN{ E6POS: X 785.5523, Y -36.1965, Z -108.0150, A 0, B 90, C 0, E1 0, E2 0, E3 0, E4 0 } C_DIS
LIN{ E6POS: X 785.6937, Y -37.1864, Z -108.0150, A 0, B 90, C 0, E1 0, E2 0, E3 0, E4 0 } C_DIS
LIN{ E6POS: X 785.7979, Y -37.9159, Z -108.0150, A 0, B 90, C 0, E1 0, E2 0, E3 0, E4 0 } C_DIS
LIN{ E6POS: X 785.9393, Y -38.9058, Z -108.0150, A 0, B 90, C 0, E1 0, E2 0, E3 0, E4 0 } C_DIS
LIN{ E6POS: X 786.0807, Y -39.8958, Z -108.0150, A 0, B 90, C 0, E1 0, E2 0, E3 0, E4 0 } C_DIS
LIN{ E6POS: X 786.1747, Y -40.5536, Z -108.0150, A 0, B 90, C 0, E1 0, E2 0, E3 0, E4 0 } C_DIS
LIN{ E6POS: X 786.0743, Y -41.5485, Z -108.0150, A 0, B 90, C 0, E1 0, E2 0, E3 0, E4 0 } C_DIS
LIN{ E6POS: X 785.9740, Y -42.5435, Z -108.0150, A 0, B 90, C 0, E1 0, E2 0, E3 0, E4 0 } C_DIS
LIN{ E6POS: X 785.8737, Y -43.5384, Z -108.0150, A 0, B 90, C 0, E1 0, E2 0, E3 0, E4 0 } C_DIS
LIN{ E6POS: X 785.7734, Y -44.5334, Z -108.0150, A 0, B 90, C 0, E1 0, E2 0, E3 0, E4 0 } C_DIS
LIN{ E6POS: X 785.6731, Y -45.5283, Z -108.0150, A 0, B 90, C 0, E1 0, E2 0, E3 0, E4 0 } C_DIS
LIN{ E6POS: X 785.5728, Y -46.5233, Z -108.0150, A 0, B 90, C 0, E1 0, E2 0, E3 0, E4 0 } C_DIS
LIN{ E6POS: X 785.4725, Y -47.5183, Z -108.0150, A 0, B 90, C 0, E1 0, E2 0, E3 0, E4 0 } C_DIS
LIN{ E6POS: X 785.3721, Y -48.5132, Z -108.0150, A 0, B 90, C 0, E1 0, E2 0, E3 0, E4 0 } C_DIS
LIN{ E6POS: X 785.3381, Y -48.8511, Z -108.0150, A 0, B 90, C 0, E1 0, E2 0, E3 0, E4 0 } C_DIS
LIN{ E6POS: X 785.2378, Y -49.8460, Z -108.0150, A 0, B 90, C 0, E1 0, E2 0, E3 0, E4 0 } C_DIS
LIN{ E6POS: X 785.1374, Y -50.8410, Z -108.0150, A 0, B 90, C 0, E1 0, E2 0, E3 0, E4 0 } C_DIS
LIN{ E6POS: X 785.0371, Y -51.8360, Z -108.0150, A 0, B 90, C 0, E1 0, E2 0, E3 0, E4 0 } C_DIS
LIN{ E6POS: X 784.9368, Y -52.8309, Z -108.0150, A 0, B 90, C 0, E1 0, E2 0, E3 0, E4 0 } C_DIS
LIN{ E6POS: X 784.8675, Y -53.5185, Z -108.0150, A 0, B 90, C 0, E1 0, E2 0, E3 0, E4 0 } C_DIS
LIN{ E6POS: X 784.6915, Y -54.5029, Z -108.0150, A 0, B 90, C 0, E1 0, E2 0, E3 0, E4 0 } C_DIS
